ABB RobotStudio station: Train_assembly_setup_60.rsstn

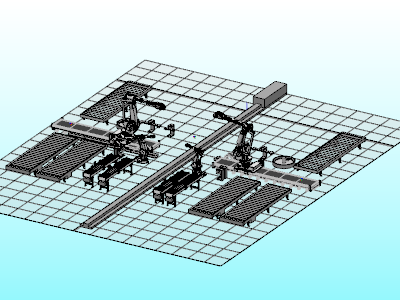
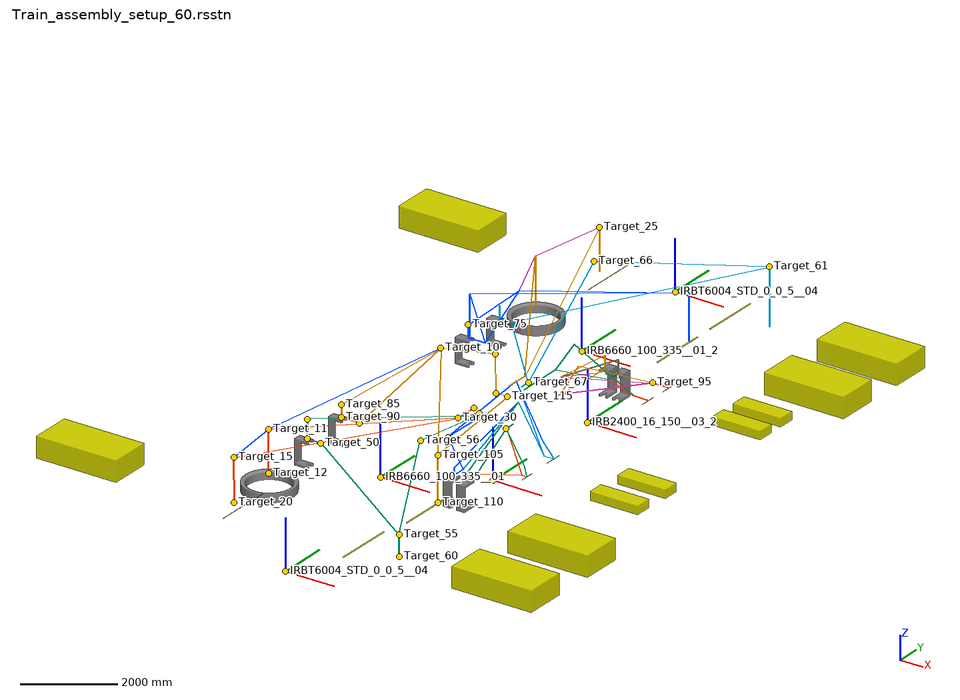
[picture v1: parts stored in the station drawn from their meshes, with robot base, taught points and paths (robot models come from the ABB library and are not in the file)]
Station Train_assembly_setup_60 (saved by RobotStudio 24.3.10958.1)
Controller Controller19, task T_ROB2: task frame (RAPID world) sits at (6880.03, 7396.16, 384.5) mm, rotated rx 0 ry 0 rz -90 deg in the station
Controller Controller19, task T_ROB1: task frame (RAPID world) sits at (6880.03, 7396.16, 384.5) mm, rotated rx 0 ry 0 rz -90 deg in the station
Controller Controller18, task T_ROB2: task frame (RAPID world) sits at (6882.77, -6739.06, 384.5) mm, rotated rx 0 ry 0 rz 90 deg in the station
Controller Controller18, task T_ROB1: task frame (RAPID world) sits at (6882.77, -6739.06, 384.5) mm, rotated rx 0 ry 0 rz 90 deg in the station
Controller Controller18
  mechanical unit ROB_1: IRB6660_100_335__01, 6 joints, base frame (0, 0, 0) mm
  mechanical unit TRACK_1: IRBT6004_STD_0_0_5__04, 1 joints, base frame (0, 0, 0) mm
  mechanical unit ROB_2: IRB2400_16_150__03, 6 joints, base frame (5338.88, -1522.95, -384.5) mm, rotated rx 0 ry 0 rz 0.09 deg
Controller Controller19
  mechanical unit ROB_1: IRB6660_100_335__01_2, 6 joints, base frame (0, 0, 0) mm
  mechanical unit TRACK_1: IRBT6004_STD_0_0_5__04_2, 1 joints, base frame (0, 0, 0) mm
  mechanical unit ROB_2: IRB2400_16_150__03_2, 6 joints, base frame (5457.45, 1561.32, -384.5) mm, rotated rx 0 ry 0 rz -0.15 deg
Layout (positions relative to the parent item):
  - train_body [part] at (-4902.1, 350, 1462.39) mm, rotated rx 90 ry 0 rz 90 deg, size 1000 x 1362.5 x 2750 mm
  - IRB6660_100_335__01 [mechanism, from %ABB.RobotStudio.Models.IRB6660%\IRB6660_100_335_G_01.rslib] at (6882.77, -3243.33, 384.5) mm, rotated rx 0 ry 0 rz 90 deg; joint values [0.0868, -0.0685, 0.1058, 0, 0.4178, 1.215] (rad or m)
  - IRBT6004_STD_0_0_5__04 [mechanism] at (7357.77, -7329.56, 0) mm, rotated rx 0 ry 0 rz 90 deg; joint values [3.4957] (rad or m)
      links: Base, Link1
  - IRB2400_16_150__03 [mechanism, from %ABB.RobotStudio.Models.IRB2400%\IRB2400_16_150_G_03.rslib] at (8405.72, -1400.18, 0) mm, rotated rx 0 ry 0 rz 90.09 deg; joint values [0, -0.2615, -0.2111, 0, 0.7347, 0] (rad or m)
  - toolHolder_2 [part] at (8688, -2615.24, 0) mm, rotated rx 0 ry 0 rz 180 deg, size 200 x 350 x 600 mm
  - toolHolder_3 [part] at (8343.34, -2615.24, 0) mm, rotated rx 0 ry 0 rz 180 deg, size 200 x 350 x 600 mm
  - toolHolder_5 [part] at (4986.26, -1820.5, 17.28) mm, rotated rx 0 ry 0 rz 90 deg, size 200 x 350 x 600 mm
  - toolHolder_6 [part] at (4986.26, -3034.43, 0) mm, rotated rx 0 ry 0 rz 90 deg, size 200 x 350 x 600 mm
  - Axel_pin [part] at (11460.69, -1282, 854.82) mm, size 562.7 x 211 x 211 mm
  - ToolHolder(wheel) [part] at (4900.07, -4399.05, 0) mm, size 1200 x 1193.4 x 200 mm
  - 1320_4800_h2 [part, from %ABB.RobotStudio.Models.Conveyors%\Conveyor 1320 4800 h2.rslib] at (701.25, 6246.74, 0) mm
  - 1320_4800_2 [part, from %ABB.RobotStudio.Models.Conveyors%\Conveyor 1320 4800 h2.rslib] at (13264.62, -5495.83, 0) mm, rotated rx 0 ry 0 rz 180 deg
  - 1320_4800_3 [part, from %ABB.RobotStudio.Models.Conveyors%\Conveyor 1320 4800 h2.rslib] at (13264.62, -3687.06, 0) mm, rotated rx 0 ry 0 rz 180 deg
  - Stack_tutorial_2 [part] at (8828.86, 5027.59, 1315.99) mm, rotated rx -90 ry 0 rz 0 deg, size 625 x 875 x 623.8 mm
  - Cow_Catcher [part] at (13797.89, -3839.41, 450.44) mm, rotated rx 0 ry 0 rz -90 deg, size 900 x 562.5 x 375 mm
  - Link [part] at (13394.81, -6331.06, 437.55) mm, rotated rx 90 ry 0 rz -90 deg, size 186.8 x 62.5 x 1937.5 mm
  - Arm_pin [part] at (10630.82, -2218.47, 824.2) mm, rotated rx 0 ry 0 rz 90 deg, size 126 x 162.5 x 125.8 mm
  - 400_guide [part, from %ABB.RobotStudio.Models.Conveyors%\Conveyor Guide 400.rslib] at (12859.46, 2271.9, 0) mm, rotated rx 0 ry 0 rz 180 deg
  - 400 [part, from %ABB.RobotStudio.Models.Conveyors%\Conveyor Guide 400.rslib] at (12859.46, -2034.23, 0) mm, rotated rx 0 ry 0 rz 180 deg
  - ZugSchlitten [mechanism] at (-2951.59, 0, 0) mm; joint values [0] (rad or m)
      links: L1, L2
  - MoveTrain_Wheel1 [smart component]
      signals: DI GetToWheel1
      connections:
        MoveTrain_Wheel1.GetToWheel1 -> PoseMover.Execute
    - PoseMover [smart component, from Components\PoseMover.rslib]
        properties: Mechanism=ZugSchlitten; Pose=2; Duration=2
  - Wheel_tool_smart [smart component] at (4882.6, -4404, 384.25) mm, rotated rx 180 ry 0 rz -0.66 deg
      signals: DI Wheel_Attach, DO Wheel_is_attached, DI findLocomotive
      connections:
        Attacher.Executed -> Wheel_tool_smart.Wheel_is_attached
        Wheel_tool_smart.Wheel_Attach -> LogicGate.InputA
        LogicGate.Output -> Detacher.Execute
        Attacher.Executed -> SetParent_2.Execute
        Detacher.Executed -> SetParent_3.Execute
        Detacher.Executed -> Attacher_2.Execute
        Wheel_tool_smart.Wheel_Attach -> ClosestObject.Execute
        ClosestObject.Executed -> Attacher.Execute
        Wheel_tool_smart.Wheel_Attach -> ClosestObject_2.Execute
        Attacher.Child => Detacher.Child
        Attacher.Child => SetParent_2.Child
        Attacher.Child => SetParent_3.Child
        Detacher.Child => Attacher_2.Child
        ClosestObject.ClosestObject => Attacher.Child
        ClosestObject.ReferenceObject => Attacher.Parent
        ClosestObject_2.ClosestObject => Attacher_2.Parent
    - WheelTool [mechanism] at (0, 0, 0) mm
        TCP WheelTool at (0, 0, 380) mm
        links: Tool_Wheel
    - Attacher [smart component, from Components\Attacher.rslib]
        properties: Parent=WheelTool; Flange=0; Child=Link_Tool_smart; Mount=false; Offset=[0 0 0]; Orientation=[0 0 0]
    - LogicGate [smart component, from Components\LogicGate.rslib]
        properties: Operator=NOT; Delay=0
    - Detacher [smart component, from Components\Detacher.rslib]
        properties: Child=Link_Tool_smart; KeepPosition=true
    - Attacher_2 [smart component, from Components\Attacher.rslib]
        properties: Parent=train_body; Flange=0; Child=Link_Tool_smart; Mount=false; Offset=[0 0 0]; Orientation=[0 0 0]
    - ClosestObject [smart component, from Components\ClosestObject.rslib]
        properties: ReferenceObject=Wheel_tool_smart; ReferencePoint=[0 0 0]; RootObject=(none); ClosestObject=Link_Tool_smart; ClosestPart=Tool_Link; Distance=0.444833038330078
    - ClosestObject_2 [smart component, from Components\ClosestObject.rslib]
        properties: ReferenceObject=L2; ReferencePoint=[0 0 0]; RootObject=(none); ClosestObject=train_body; ClosestPart=train_body; Distance=0
  - Wheel [part] at (3497.77, -6177.47, 411.44) mm, size 1122.9 x 1119.7 x 250 mm
  - Axel_Tool_smart [smart component] at (8343.34, -2684.49, 620.79) mm, rotated rx 180 ry 0 rz 0 deg
      signals: DI Grab_with_tool, DO partAttached
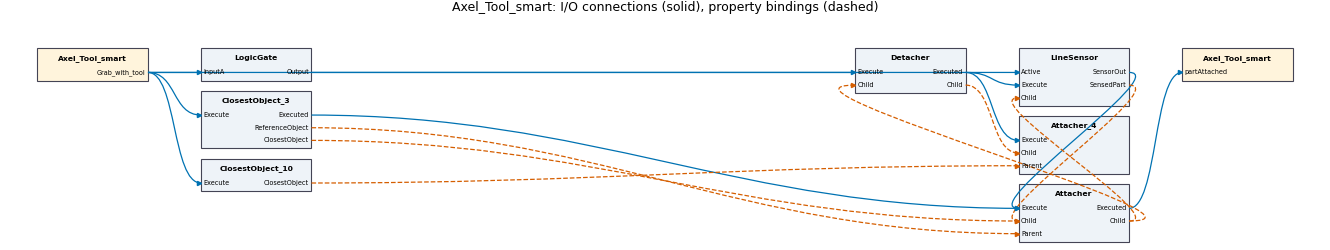
      connections:
        Axel_Tool_smart.Grab_with_tool -> LineSensor.Active
        LineSensor.SensorOut -> Attacher.Execute
        Axel_Tool_smart.Grab_with_tool -> LogicGate.InputA
        LogicGate.Output -> Detacher.Execute
        Detacher.Executed -> SetParent_4.Execute
        Attacher.Executed -> Axel_Tool_smart.partAttached
        Axel_Tool_smart.Grab_with_tool -> ClosestObject_3.Execute
        ClosestObject_3.Executed -> Attacher.Execute
        Detacher.Executed -> Attacher_4.Execute
        Axel_Tool_smart.Grab_with_tool -> ClosestObject_10.Execute
        LineSensor.SensedPart => Attacher.Child
        Attacher.Child => Detacher.Child
        Attacher.Child => SetParent_4.Child
        ClosestObject_3.ReferenceObject => Attacher.Parent
        ClosestObject_3.ClosestObject => Attacher.Child
        Detacher.Child => Attacher_4.Child
        ClosestObject_10.ClosestObject => Attacher_4.Parent
    - AxelTool [mechanism] at (0, 9.42, 0) mm
        TCP AxelTool at (0, 0, 262.49) mm
        links: Tool_Axel_pin
    - Detacher [smart component, from Components\Detacher.rslib]
        properties: Child=Pin_Tool_smart; KeepPosition=true
    - LogicGate [smart component, from Components\LogicGate.rslib]
        properties: Operator=NOT; Delay=0
    - Attacher [smart component, from Components\Attacher.rslib]
        properties: Parent=Axel_Tool_smart; Flange=0; Child=Pin_Tool_smart; Mount=false; Offset=[0 0 0]; Orientation=[0 0 0]
    - ClosestObject_3 [smart component, from Components\ClosestObject.rslib]
        properties: ReferenceObject=Axel_Tool_smart; ReferencePoint=[0 0 0]; RootObject=(none); ClosestObject=Pin_Tool_smart; ClosestPart=Tool_Arm_pin; Distance=0.139682907104492
    - Attacher_4 [smart component, from Components\Attacher.rslib]
        properties: Parent=(none); Flange=0; Child=Pin_Tool_smart; Mount=false; Offset=[0 0 0]; Orientation=[0 0 0]
    - ClosestObject_10 [smart component, from Components\ClosestObject.rslib]
        properties: ReferenceObject=L2; ReferencePoint=[0 0 0]; RootObject=(none); ClosestObject=(none); ClosestPart=(none); Distance=0
  - AttachTool_Rob1 [smart component] at (6695.48, -1090.62, 2469) mm, rotated rx 121.63 ry 17.56 rz -164.5 deg
      signals: DI AttachTool, DO ToolAttached
      connections:
        AttachTool_Rob1.AttachTool -> ClosestObject.Execute
        ClosestObject.Executed -> Attacher.Execute
        AttachTool_Rob1.AttachTool -> LogicGate.InputA
        LogicGate.Output -> Detacher.Execute
        Attacher.Executed -> AttachTool_Rob1.ToolAttached
        ClosestObject.ClosestObject => Attacher.Child
        Attacher.Child => Detacher.Child
    - ClosestObject [smart component, from Components\ClosestObject.rslib]
        properties: ReferenceObject=IRB6660_100_335__01; ReferencePoint=[7.13389 -0.654994 0.85]; RootObject=(none); ClosestObject=Axel_Tool_smart; ClosestPart=Tool_Axel_pin; Distance=0.924461853027344
    - Attacher [smart component, from Components\Attacher.rslib]
        properties: Parent=IRB6660_100_335__01; Flange=0; Child=Axel_Tool_smart; Mount=false; Offset=[0 0 0]; Orientation=[0 0 0]
    - LogicGate [smart component, from Components\LogicGate.rslib]
        properties: Operator=NOT; Delay=0
    - Detacher [smart component, from Components\Detacher.rslib]
        properties: Child=Axel_Tool_smart; KeepPosition=true
  - AttachTool_Rob2 [smart component] at (8404.6, -698.88, 1543.74) mm, rotated rx 180 ry 60 rz -89.91 deg
      signals: DI AttachTool, DO ToolAttached
      connections:
        AttachTool_Rob2.AttachTool -> ClosestObject.Execute
        ClosestObject.Executed -> Attacher.Execute
        AttachTool_Rob2.AttachTool -> LogicGate.InputA
        LogicGate.Output -> Detacher.Execute
        Attacher.Executed -> AttachTool_Rob2.ToolAttached
        ClosestObject.ClosestObject => Attacher.Child
        Attacher.Child => Detacher.Child
    - ClosestObject [smart component, from Components\ClosestObject.rslib]
        properties: ReferenceObject=IRB2400_16_150__03; ReferencePoint=[7.483895 -1.376883 0.85]; RootObject=(none); ClosestObject=Axel_Tool_smart; ClosestPart=Tool_Axel_pin; Distance=0.745236877441406
    - Attacher [smart component, from Components\Attacher.rslib]
        properties: Parent=IRB2400_16_150__03; Flange=0; Child=Axel_Tool_smart; Mount=false; Offset=[0 0 0]; Orientation=[0 0 0]
    - LogicGate [smart component, from Components\LogicGate.rslib]
        properties: Operator=NOT; Delay=0
    - Detacher [smart component, from Components\Detacher.rslib]
        properties: Child=Axel_Tool_smart; KeepPosition=true
  - MoveTrain_Wheel2 [smart component]
      signals: DI GetToWheel2
      connections:
        MoveTrain_Wheel2.GetToWheel2 -> PoseMover.Execute
    - PoseMover [smart component, from Components\PoseMover.rslib]
        properties: Mechanism=ZugSchlitten; Pose=3; Duration=1
  - Locomotive [smart component] at (-3926.39, 500, 862.39) mm
  - SpawnWheel [smart component]
      signals: DO volumeerkannt, DI spanw, DI diDeque
      connections:
        VolumeSensor.SensorOut -> LogicGate.InputA
        LineSensor_2.SensorOut -> LogicGate_2.InputA
        LogicGate_2.Output -> LinearMover.Execute
        Source.Executed -> Queue_2.Enqueue
        LogicGate.Output -> Source.Execute
        SpawnWheel.diDeque -> Queue_2.Dequeue
        SpawnWheel.spanw -> Source.Execute
        Source.Copy => Queue_2.Back
    - Source [smart component, from Components\Source.rslib]
        properties: Source=Wheel; Copy=(none); Parent=(none); Position=[1.2 -6.177465 0.41144]; Orientation=[0 0 0]; Transient=false; PhysicsBehavior=-1
    - Queue_2 [smart component, from Components\Queue.rslib]
        properties: Back=(none); Front=(none); Queue={1d260e56-3a9b-4089-bc8a-9b7fc13f89e8};{5a10ac6e-8e6d-4320-b1fc-87ca64eb2ab9}; NumberOfObjects=2
    - LinearMover [smart component, from Components\LinearMover.rslib]
        properties: Object=Queue_2; Direction=[1 0 0]; Speed=0.8; Reference=Global; ReferenceObject=(none)
    - LineSensor_2 [smart component, from Components\LineSensor.rslib]
        properties: Start=[5.47 -6.89178 0.5]; End=[5.47 -5.45178 0.5]; Length=1.44; Radius=0.00524017467248908; Tag=(none); SensedPart=(none); SensedPoint=[0 0 0]
      - _sensorPart_ [part], size 10.5 x 1440 x 10.5 mm
    - VolumeSensor [smart component, from Components\VolumeSensor.rslib]
        properties: CornerPoint=[0.761246 -6.83178 0.55]; Orientation=[0 0 0]; Length=2; Width=1; Height=0.5; Tag=(none); PartialHit=true; SensedPart=(none)
      - _sensorPart_ [part], size 2000 x 1000 x 500 mm
    - LogicGate [smart component, from Components\LogicGate.rslib]
        properties: Operator=NOT; Delay=0
    - LogicGate_2 [smart component, from Components\LogicGate.rslib]
        properties: Operator=NOT; Delay=0
  - SpawnAxel [smart component]
      signals: DO volumeerkannt, DI spanw, DI diDeque
      connections:
        VolumeSensor.SensorOut -> LogicGate.InputA
        LineSensor_2.SensorOut -> LogicGate_2.InputA
        LogicGate_2.Output -> LinearMover.Execute
        Source.Executed -> Queue_2.Enqueue
        LogicGate.Output -> Source.Execute
        SpawnAxel.diDeque -> Queue_2.Dequeue
        Source.Copy => Queue_2.Back
    - Source [smart component, from Components\Source.rslib]
        properties: Source=Axel_pin; Copy=(none); Parent=(none); Position=[12.5 -1.280871 0.854819]; Orientation=[0 0 0]; Transient=false; PhysicsBehavior=-1
    - Queue_2 [smart component, from Components\Queue.rslib]
        properties: Back=(none); Front=(none); Queue={1d260e56-3a9b-4089-bc8a-9b7fc13f89e8}; NumberOfObjects=1
    - LinearMover [smart component, from Components\LinearMover.rslib]
        properties: Object=Queue_2; Direction=[-1 0 0]; Speed=0.5; Reference=Global; ReferenceObject=(none)
    - LineSensor_2 [smart component, from Components\LineSensor.rslib]
        properties: Start=[9.859459 -1.543182 0.86]; End=[9.859459 -1.100182 0.86]; Length=0.443; Radius=0.00524017467248908; Tag=(none); SensedPart=(none); SensedPoint=[0 0 0]
      - _sensorPart_ [part], size 10.5 x 443 x 10.5 mm
    - VolumeSensor [smart component, from Components\VolumeSensor.rslib]
        properties: CornerPoint=[11.6 -1.5 0.86]; Orientation=[0 0 0]; Length=1.2; Width=0.4; Height=0.2; Tag=(none); PartialHit=true; SensedPart=(none)
      - _sensorPart_ [part], size 1200 x 400 x 200 mm
    - LogicGate [smart component, from Components\LogicGate.rslib]
        properties: Operator=NOT; Delay=0
    - LogicGate_2 [smart component, from Components\LogicGate.rslib]
        properties: Operator=NOT; Delay=0
  - IRB2400_16_150__03_2 [mechanism, from %ABB.RobotStudio.Models.IRB2400%\IRB2400_16_150_G_03.rslib] at (8441.35, 1938.71, 0) mm, rotated rx 0 ry 0 rz -90.15 deg; joint values [0, -0.2615, -0.2111, 0, 0.7347, 0] (rad or m)
  - IRBT6004_STD_0_0_5__04_2 [mechanism] at (6405.03, 7986.66, 0) mm, rotated rx 0 ry 0 rz -90 deg; joint values [3.4275] (rad or m)
      links: Base, Link1
  - IRB6660_100_335__01_2 [mechanism, from %ABB.RobotStudio.Models.IRB6660%\IRB6660_100_335_G_01.rslib] at (6880.03, 3968.65, 384.5) mm, rotated rx 0 ry 0 rz -90 deg; joint values [0, -0.2199, -0.1274, 0, 0.651, 0] (rad or m)
  - 1320_4800_4 [part, from %ABB.RobotStudio.Models.Conveyors%\Conveyor 1320 4800 h2.rslib] at (701.25, -6831.78, 0) mm
  - ToolHolder(wheel)_2 [part] at (4900.07, 5155.46, 0) mm, size 1200 x 1193.4 x 200 mm
  - toolHolder_7 [part] at (4986.26, 3849.13, 0) mm, rotated rx 0 ry 0 rz 90 deg, size 200 x 350 x 600 mm
  - toolHolder_8 [part] at (4986.26, 2721.93, 17.28) mm, rotated rx 0 ry 0 rz 90 deg, size 200 x 350 x 600 mm
  - Wheel_tool_smart_2 [smart component] at (4882.6, 5151.99, 384.25) mm, rotated rx -180 ry 0 rz -0.66 deg
      signals: DI Wheel_Attach, DO Wheel_is_attached
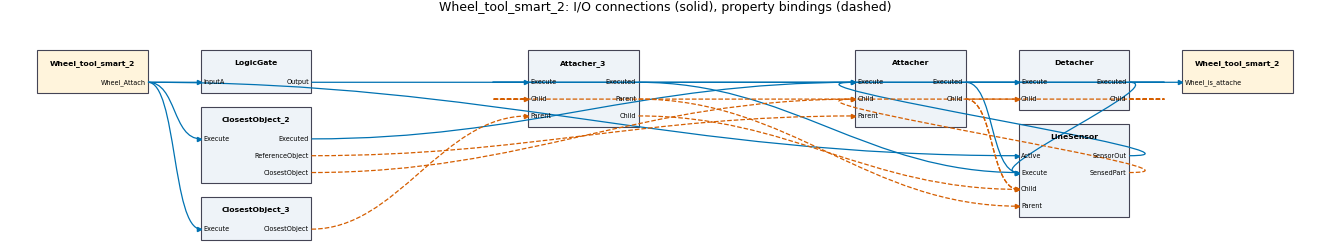
      connections:
        Wheel_tool_smart_2.Wheel_Attach -> LineSensor.Active
        LineSensor.SensorOut -> Attacher.Execute
        Attacher.Executed -> Wheel_tool_smart_2.Wheel_is_attached
        Wheel_tool_smart_2.Wheel_Attach -> LogicGate.InputA
        LogicGate.Output -> Detacher.Execute
        Attacher.Executed -> ?.Execute
        Detacher.Executed -> SetParent_3.Execute
        Wheel_tool_smart_2.Wheel_Attach -> ClosestObject_2.Execute
        ClosestObject_2.Executed -> Attacher.Execute
        Detacher.Executed -> Attacher_3.Execute
        Wheel_tool_smart_2.Wheel_Attach -> ClosestObject_3.Execute
        Attacher_3.Executed -> SetParent.Execute
        LineSensor.SensedPart => Attacher.Child
        Attacher.Child => Detacher.Child
        Attacher.Child => ?.Child
        Attacher.Child => SetParent_3.Child
        ClosestObject_2.ReferenceObject => Attacher.Parent
        ClosestObject_2.ClosestObject => Attacher.Child
        Detacher.Child => Attacher_3.Child
        ClosestObject_3.ClosestObject => Attacher_3.Parent
        Attacher_3.Parent => SetParent.Parent
        Attacher_3.Child => SetParent.Child
    - WheelTool [mechanism] at (11.79, -0.14, 0) mm
        TCP WheelTool at (0, 0, 380) mm
        links: Tool_Wheel
    - Attacher [smart component, from Components\Attacher.rslib]
        properties: Parent=WheelTool; Flange=0; Child=Link_Tool_smart_2; Mount=false; Offset=[0 0 0]; Orientation=[0 0 0]
    - LogicGate [smart component, from Components\LogicGate.rslib]
        properties: Operator=NOT; Delay=0
    - Detacher [smart component, from Components\Detacher.rslib]
        properties: Child=Link_Tool_smart_2; KeepPosition=true
    - ClosestObject_2 [smart component, from Components\ClosestObject.rslib]
        properties: ReferenceObject=Wheel_tool_smart_2; ReferencePoint=[0 0 0]; RootObject=(none); ClosestObject=Link_Tool_smart_2; ClosestPart=Tool_Link; Distance=0.391564422607422
    - Attacher_3 [smart component, from Components\Attacher.rslib]
        properties: Parent=train_body; Flange=0; Child=Link_Tool_smart_2; Mount=false; Offset=[0 0 0]; Orientation=[0 0 0]
    - ClosestObject_3 [smart component, from Components\ClosestObject.rslib]
        properties: ReferenceObject=L2; ReferencePoint=[0 0 0]; RootObject=(none); ClosestObject=train_body; ClosestPart=train_body; Distance=1.51384008789063
  - toolHolder_10 [part] at (8343.34, 3102.04, 0) mm, size 200 x 350 x 600 mm
  - 400_2 [part, from %ABB.RobotStudio.Models.Conveyors%\Conveyor Guide 400.rslib] at (12859.46, -1103.18, 0) mm, rotated rx 0 ry 0 rz 180 deg
  - SpawnAxel_2 [smart component]
      signals: DO volumeerkannt, DI spanw, DI diDeque
      connections:
        VolumeSensor.SensorOut -> LogicGate.InputA
        LineSensor_2.SensorOut -> LogicGate_2.InputA
        LogicGate_2.Output -> LinearMover.Execute
        Source.Executed -> Queue_2.Enqueue
        LogicGate.Output -> Source.Execute
        SpawnAxel_2.diDeque -> Queue_2.Dequeue
        SpawnAxel_2.spanw -> Source.Execute
        VolumeSensor.SensorOut -> SpawnAxel_2.volumeerkannt
        Source.Copy => Queue_2.Back
    - Source [smart component, from Components\Source.rslib]
        properties: Source=Axel_pin_2; Copy=(none); Parent=(none); Position=[12.5 2.071151 0.854819]; Orientation=[0 0 0]; Transient=false; PhysicsBehavior=-1
    - Queue_2 [smart component, from Components\Queue.rslib]
        properties: Back=(none); Front=(none); Queue={1d260e56-3a9b-4089-bc8a-9b7fc13f89e8};{68ae6273-f876-46ed-a841-c22bc3c7f170}; NumberOfObjects=1
    - LinearMover [smart component, from Components\LinearMover.rslib]
        properties: Object=Queue_2; Direction=[-1 0 0]; Speed=0.5; Reference=Global; ReferenceObject=(none)
    - LineSensor_2 [smart component, from Components\LineSensor.rslib]
        properties: Start=[9.859459 1.8769 0.84]; End=[9.859459 2.2749 0.84]; Length=0.398; Radius=0.00524017467248908; Tag=(none); SensedPart=(none); SensedPoint=[0 0 0]
      - _sensorPart_ [part], size 10.5 x 398 x 10.5 mm
    - VolumeSensor [smart component, from Components\VolumeSensor.rslib]
        properties: CornerPoint=[11.617459 1.8719 0.86]; Orientation=[0 0 0]; Length=1.2; Width=0.4; Height=0.2; Tag=(none); PartialHit=true; SensedPart=(none)
      - _sensorPart_ [part], size 1200 x 400 x 200 mm
    - LogicGate [smart component, from Components\LogicGate.rslib]
        properties: Operator=NOT; Delay=0
    - LogicGate_2 [smart component, from Components\LogicGate.rslib]
        properties: Operator=NOT; Delay=0
  - Axel_pin_2 [part] at (11364, 2071.15, 854.82) mm, size 562.7 x 211 x 211 mm
  - Axel_Tool_smart_2 [smart component] at (8343.34, 3189.01, 620.79) mm, rotated rx 180 ry 0 rz 0 deg
      signals: DI Grab_with_tool, DO partAttached
      connections:
        Axel_Tool_smart_2.Grab_with_tool -> LineSensor.Active
        LineSensor.SensorOut -> Attacher.Execute
        Axel_Tool_smart_2.Grab_with_tool -> LogicGate.InputA
        LogicGate.Output -> Detacher.Execute
        Detacher.Executed -> SetParent_4.Execute
        Attacher.Executed -> Axel_Tool_smart_2.partAttached
        Axel_Tool_smart_2.Grab_with_tool -> ClosestObject_4.Execute
        ClosestObject_4.Executed -> Attacher.Execute
        Detacher.Executed -> Attacher_5.Execute
        Axel_Tool_smart_2.Grab_with_tool -> ClosestObject_11.Execute
        LineSensor.SensedPart => Attacher.Child
        Attacher.Child => Detacher.Child
        Attacher.Child => SetParent_4.Child
        ClosestObject_4.ReferenceObject => Attacher.Parent
        ClosestObject_4.ClosestObject => Attacher.Child
        Detacher.Child => Attacher_5.Child
        ClosestObject_11.ClosestObject => Attacher_5.Parent
    - AxelTool [mechanism] at (0, 9.42, 0) mm
        TCP AxelTool at (0, 0, 262.49) mm
        links: Tool_Axel_pin
    - Detacher [smart component, from Components\Detacher.rslib]
        properties: Child=toolHolder_10; KeepPosition=true
    - LogicGate [smart component, from Components\LogicGate.rslib]
        properties: Operator=NOT; Delay=0
    - Attacher [smart component, from Components\Attacher.rslib]
        properties: Parent=Axel_Tool_smart_2; Flange=0; Child=toolHolder_10; Mount=false; Offset=[0 0 0]; Orientation=[0 0 0]
    - ClosestObject_4 [smart component, from Components\ClosestObject.rslib]
        properties: ReferenceObject=Axel_Tool_smart_2; ReferencePoint=[0 0 0]; RootObject=(none); ClosestObject=toolHolder_10; ClosestPart=toolHolder_10; Distance=0
    - Attacher_5 [smart component, from Components\Attacher.rslib]
        properties: Parent=train_body; Flange=0; Child=toolHolder_10; Mount=false; Offset=[0 0 0]; Orientation=[0 0 0]
    - ClosestObject_11 [smart component, from Components\ClosestObject.rslib]
        properties: ReferenceObject=L2; ReferencePoint=[0 0 0]; RootObject=(none); ClosestObject=train_body; ClosestPart=train_body; Distance=1.51384008789063
  - AttachTool_Rob4 [smart component] at (8508.36, -848.72, 1842.51) mm, rotated rx 14.33 ry -9.97 rz 155.57 deg
      signals: DI AttachTool, DO ToolAttached
      connections:
        AttachTool_Rob4.AttachTool -> ClosestObject.Execute
        ClosestObject.Executed -> Attacher.Execute
        AttachTool_Rob4.AttachTool -> LogicGate.InputA
        LogicGate.Output -> Detacher.Execute
        Attacher.Executed -> AttachTool_Rob4.ToolAttached
        ClosestObject.ClosestObject => Attacher.Child
        Attacher.Child => Detacher.Child
    - ClosestObject [smart component, from Components\ClosestObject.rslib]
        properties: ReferenceObject=IRB2400_16_150__03_2; ReferencePoint=[7.483895 1.442587 0.85]; RootObject=(none); ClosestObject=toolHolder_10; ClosestPart=toolHolder_10; Distance=0.689487548828125
    - Attacher [smart component, from Components\Attacher.rslib]
        properties: Parent=IRB2400_16_150__03_2; Flange=0; Child=toolHolder_10; Mount=false; Offset=[0 0 0]; Orientation=[0 0 0]
    - LogicGate [smart component, from Components\LogicGate.rslib]
        properties: Operator=NOT; Delay=0
    - Detacher [smart component, from Components\Detacher.rslib]
        properties: Child=toolHolder_10; KeepPosition=true
  - AttachTool_Rob3 [smart component] at (8508.36, -848.72, 1842.51) mm, rotated rx 14.33 ry -9.97 rz 155.57 deg
      signals: DI AttachTool, DO ToolAttached
      connections:
        AttachTool_Rob3.AttachTool -> ClosestObject.Execute
        ClosestObject.Executed -> Attacher.Execute
        AttachTool_Rob3.AttachTool -> LogicGate.InputA
        LogicGate.Output -> Detacher.Execute
        Attacher.Executed -> AttachTool_Rob3.ToolAttached
        ClosestObject.ClosestObject => Attacher.Child
        Attacher.Child => Detacher.Child
    - ClosestObject [smart component, from Components\ClosestObject.rslib]
        properties: ReferenceObject=IRB6660_100_335__01_2; ReferencePoint=[4.894392 5.151995 0.65291]; RootObject=(none); ClosestObject=Pin_Tool_smart2; ClosestPart=Tool_Arm_pin; Distance=0.77755078125
    - Attacher [smart component, from Components\Attacher.rslib]
        properties: Parent=IRB6660_100_335__01_2; Flange=0; Child=Pin_Tool_smart2; Mount=false; Offset=[0 0 0]; Orientation=[0 0 0]
    - LogicGate [smart component, from Components\LogicGate.rslib]
        properties: Operator=NOT; Delay=0
    - Detacher [smart component, from Components\Detacher.rslib]
        properties: Child=Pin_Tool_smart2; KeepPosition=true
  - Wheel_2 [part] at (3426.57, 6899.85, 411.8) mm, size 1122.9 x 1119.7 x 250 mm
  - SpawnWheel_2 [smart component]
      signals: DO volumeerkannt, DI spanw, DI diDeque
      connections:
        VolumeSensor.SensorOut -> LogicGate.InputA
        LineSensor_2.SensorOut -> LogicGate_2.InputA
        LogicGate_2.Output -> LinearMover.Execute
        Source.Executed -> Queue_2.Enqueue
        LogicGate.Output -> Source.Execute
        SpawnWheel_2.diDeque -> Queue_2.Dequeue
        SpawnWheel_2.spanw -> Source.Execute
        Source.Copy => Queue_2.Back
    - Source [smart component, from Components\Source.rslib]
        properties: Source=Wheel_2; Copy=(none); Parent=(none); Position=[1.8 6.899851 0.411803]; Orientation=[0 0 0]; Transient=false; PhysicsBehavior=-1
    - Queue_2 [smart component, from Components\Queue.rslib]
        properties: Back=(none); Front=(none); Queue={1d260e56-3a9b-4089-bc8a-9b7fc13f89e8}; NumberOfObjects=1
    - LinearMover [smart component, from Components\LinearMover.rslib]
        properties: Object=Queue_2; Direction=[1 0 0]; Speed=0.8; Reference=Global; ReferenceObject=(none)
    - LineSensor_2 [smart component, from Components\LineSensor.rslib]
        properties: Start=[5.47 6.186738 0.5]; End=[5.47 7.626738 0.5]; Length=1.44; Radius=0.00524017467248908; Tag=(none); SensedPart=(none); SensedPoint=[0 0 0]
      - _sensorPart_ [part], size 10.5 x 1440 x 10.5 mm
    - VolumeSensor [smart component, from Components\VolumeSensor.rslib]
        properties: CornerPoint=[0.577246 6.4 0.471]; Orientation=[0 0 0]; Length=2; Width=1; Height=0.5; Tag=(none); PartialHit=true; SensedPart=(none)
      - _sensorPart_ [part], size 2000 x 1000 x 500 mm
    - LogicGate [smart component, from Components\LogicGate.rslib]
        properties: Operator=NOT; Delay=0
    - LogicGate_2 [smart component, from Components\LogicGate.rslib]
        properties: Operator=NOT; Delay=0
  - 1320_4800_5 [part, from %ABB.RobotStudio.Models.Conveyors%\Conveyor 1320 4800 h2.rslib] at (13264.62, 7587.02, 0) mm, rotated rx 0 ry 0 rz 180 deg
  - Link_Tool_smart [smart component]
      signals: DI Link_Attach, DO Link_is_attached
      connections:
        Link_Tool_smart.Link_Attach -> ClosestObject.Execute
        ClosestObject.Executed -> Attacher.Execute
        Link_Tool_smart.Link_Attach -> LogicGate.InputA
        LogicGate.Output -> Detacher.Execute
        Detacher.Executed -> Attacher_2.Execute
        Attacher.Executed -> Link_Tool_smart.Link_is_attached
        Link_Tool_smart.Link_Attach -> ClosestObject_4.Execute
        ClosestObject.ReferenceObject => Attacher.Parent
        ClosestObject.ClosestObject => Attacher.Child
        Attacher.Child => Detacher.Child
        Detacher.Child => Attacher_2.Child
        ClosestObject_4.ClosestObject => Attacher_2.Parent
    - LinkTool [mechanism] at (4906.26, -3034.43, 624.04) mm, rotated rx 180 ry 0 rz 0 deg
        TCP LinkTool at (0, 0, 170) mm
        links: Tool_Link
    - ClosestObject [smart component, from Components\ClosestObject.rslib]
        properties: ReferenceObject=Link_Tool_smart; ReferencePoint=[0 0 0]; RootObject=(none); ClosestObject=Wheel_tool_smart; ClosestPart=Tool_Wheel; Distance=0.444832855224609
    - Attacher [smart component, from Components\Attacher.rslib]
        properties: Parent=Link_Tool_smart; Flange=0; Child=Wheel_tool_smart; Mount=false; Offset=[0 0 0]; Orientation=[0 0 0]
    - LogicGate [smart component, from Components\LogicGate.rslib]
        properties: Operator=NOT; Delay=0
    - Detacher [smart component, from Components\Detacher.rslib]
        properties: Child=Wheel_tool_smart; KeepPosition=true
    - Attacher_2 [smart component, from Components\Attacher.rslib]
        properties: Parent=(none); Flange=0; Child=Wheel_tool_smart; Mount=false; Offset=[0 0 0]; Orientation=[0 0 0]
    - ClosestObject_4 [smart component, from Components\ClosestObject.rslib]
        properties: ReferenceObject=L2; ReferencePoint=[0 0 0]; RootObject=(none); ClosestObject=(none); ClosestPart=(none); Distance=0
  - Pin_Tool_smart [smart component]
      signals: DI AttachPin, DO Pin_Attached
      connections:
        Pin_Tool_smart.AttachPin -> ClosestObject.Execute
        ClosestObject.Executed -> Attacher.Execute
        Pin_Tool_smart.AttachPin -> LogicGate.InputA
        LogicGate.Output -> Detacher.Execute
        Detacher.Executed -> Attacher_2.Execute
        Attacher.Executed -> Pin_Tool_smart.Pin_Attached
        Pin_Tool_smart.AttachPin -> ClosestObject_8.Execute
        ClosestObject.ReferenceObject => Attacher.Parent
        ClosestObject.ClosestObject => Attacher.Child
        Attacher.Child => Detacher.Child
        Detacher.Child => Attacher_2.Child
        ClosestObject_8.ClosestObject => Attacher_2.Parent
    - PinTool [mechanism] at (8688, -2695.24, 620.9) mm, rotated rx 180 ry 0 rz 0 deg
        TCP PinTool at (0, 0, 137.35) mm
        links: Tool_Arm_pin
    - ClosestObject [smart component, from Components\ClosestObject.rslib]
        properties: ReferenceObject=Pin_Tool_smart; ReferencePoint=[0 0 0]; RootObject=(none); ClosestObject=Axel_Tool_smart; ClosestPart=Tool_Axel_pin; Distance=0.139682907104492
    - Attacher [smart component, from Components\Attacher.rslib]
        properties: Parent=Pin_Tool_smart; Flange=0; Child=Axel_Tool_smart; Mount=false; Offset=[0 0 0]; Orientation=[0 0 0]
    - LogicGate [smart component, from Components\LogicGate.rslib]
        properties: Operator=NOT; Delay=0
    - Detacher [smart component, from Components\Detacher.rslib]
        properties: Child=Axel_Tool_smart; KeepPosition=true
    - Attacher_2 [smart component, from Components\Attacher.rslib]
        properties: Parent=(none); Flange=0; Child=Axel_Tool_smart; Mount=false; Offset=[0 0 0]; Orientation=[0 0 0]
    - ClosestObject_8 [smart component, from Components\ClosestObject.rslib]
        properties: ReferenceObject=L2; ReferencePoint=[0 0 0]; RootObject=(none); ClosestObject=(none); ClosestPart=(none); Distance=0
  - MoveTrain_Pin1 [smart component]
      signals: DI Move_to_pin1
      connections:
        MoveTrain_Pin1.Move_to_pin1 -> PoseMover.Execute
    - PoseMover [smart component, from Components\PoseMover.rslib]
        properties: Mechanism=ZugSchlitten; Pose=4; Duration=1
  - SpawnPin [smart component] at (0, -400, 0) mm
      signals: DO volumeerkannt, DI spanw, DI diDeque
      connections:
        VolumeSensor.SensorOut -> LogicGate.InputA
        LineSensor_2.SensorOut -> LogicGate_2.InputA
        LogicGate_2.Output -> LinearMover.Execute
        Source.Executed -> Queue_2.Enqueue
        LogicGate.Output -> Source.Execute
        SpawnPin.diDeque -> Queue_2.Dequeue
        Source.Copy => Queue_2.Back
    - Source [smart component, from Components\Source.rslib]
        properties: Source=Arm_pin; Copy=(none); Parent=(none); Position=[12.6 -2.218466 0.824201]; Orientation=[0 0 1.5707963267949]; Transient=false; PhysicsBehavior=-1
    - Queue_2 [smart component, from Components\Queue.rslib]
        properties: Back=(none); Front=(none); Queue={1d260e56-3a9b-4089-bc8a-9b7fc13f89e8}; NumberOfObjects=1
    - LinearMover [smart component, from Components\LinearMover.rslib]
        properties: Object=Queue_2; Direction=[-1 0 0]; Speed=0.5; Reference=Global; ReferenceObject=(none)
    - LineSensor_2 [smart component, from Components\LineSensor.rslib]
        properties: Start=[9.84 -1.633232 0.82]; End=[9.84 -2 0.82]; Length=0.366768; Radius=0.00524017467248908; Tag=(none); SensedPart=(none); SensedPoint=[0 0 0]
      - _sensorPart_ [part], size 10.5 x 366.8 x 10.5 mm
    - VolumeSensor [smart component, from Components\VolumeSensor.rslib]
        properties: CornerPoint=[11.56 -2.03 0.85]; Orientation=[0 0 0]; Length=1.2; Width=0.4; Height=0.2; Tag=(none); PartialHit=true; SensedPart=(none)
      - _sensorPart_ [part], size 1200 x 400 x 200 mm
    - LogicGate [smart component, from Components\LogicGate.rslib]
        properties: Operator=NOT; Delay=0
    - LogicGate_2 [smart component, from Components\LogicGate.rslib]
        properties: Operator=NOT; Delay=0
  - SpawnLink [smart component] at (10414.69, 0, 0) mm
      signals: DO volumeerkannt, DI spanw, DI diDeque
      connections:
        VolumeSensor.SensorOut -> LogicGate.InputA
        LineSensor_2.SensorOut -> LogicGate_2.InputA
        LogicGate_2.Output -> LinearMover.Execute
        Source.Executed -> Queue_2.Enqueue
        LogicGate.Output -> Source.Execute
        SpawnLink.diDeque -> Queue_2.Dequeue
        SpawnLink.spanw -> Source.Execute
        Source.Copy => Queue_2.Back
    - Source [smart component, from Components\Source.rslib]
        properties: Source=Link; Copy=(none); Parent=(none); Position=[11.5 -6.331 0.43755]; Orientation=[1.5707963267949 0 -1.5707963267949]; Transient=false; PhysicsBehavior=-1
    - Queue_2 [smart component, from Components\Queue.rslib]
        properties: Back=(none); Front=(none); Queue={1d260e56-3a9b-4089-bc8a-9b7fc13f89e8};{5a10ac6e-8e6d-4320-b1fc-87ca64eb2ab9};{339d23b8-4dd4-4c1e-9a58-b77691da5f86}; NumberOfObjects=1
    - LinearMover [smart component, from Components\LinearMover.rslib]
        properties: Object=Queue_2; Direction=[-1 0 0]; Speed=0.5; Reference=Global; ReferenceObject=(none)
    - LineSensor_2 [smart component, from Components\LineSensor.rslib] at (-7385.86, 0, -29.99) mm
        properties: Start=[5.47 -6.89178 0.5]; End=[5.47 -5.45178 0.5]; Length=1.44; Radius=0.0131004366812227; Tag=(none); SensedPart=(none); SensedPoint=[0 0 0]
      - _sensorPart_ [part], size 26.2 x 1440 x 26.2 mm
    - VolumeSensor [smart component, from Components\VolumeSensor.rslib]
        properties: CornerPoint=[0.761246486480401 -6.83178 0.49]; Orientation=[0 0 0]; Length=2; Width=1; Height=0.5; Tag=(none); PartialHit=true; SensedPart=(none)
      - _sensorPart_ [part], size 2000 x 1000 x 500 mm
    - LogicGate [smart component, from Components\LogicGate.rslib]
        properties: Operator=NOT; Delay=0
    - LogicGate_2 [smart component, from Components\LogicGate.rslib]
        properties: Operator=NOT; Delay=0
  - MoveTrain_Pin2 [smart component]
      signals: DI Get_to_Pin2
      connections:
        MoveTrain_Pin2.Get_to_Pin2 -> PoseMover.Execute
    - PoseMover [smart component, from Components\PoseMover.rslib]
        properties: Mechanism=ZugSchlitten; Pose=5; Duration=1
  - Link_Tool_smart_2 [smart component] at (4906.26, 3849.13, 626.19) mm
      signals: DI Link_Attach, DO Link_is_attached
      connections:
        Link_Tool_smart_2.Link_Attach -> ClosestObject.Execute
        ClosestObject.Executed -> Attacher.Execute
        Link_Tool_smart_2.Link_Attach -> LogicGate.InputA
        LogicGate.Output -> Detacher.Execute
        Detacher.Executed -> Attacher_2.Execute
        Attacher.Executed -> Link_Tool_smart_2.Link_is_attached
        Link_Tool_smart_2.Link_Attach -> ClosestObject_5.Execute
        ClosestObject.ReferenceObject => Attacher.Parent
        ClosestObject.ClosestObject => Attacher.Child
        Attacher.Child => Detacher.Child
        Detacher.Child => Attacher_2.Child
        ClosestObject_5.ClosestObject => Attacher_2.Parent
    - LinkTool [mechanism] at (0, 0, 0) mm, rotated rx 180 ry 0 rz 0 deg
        TCP LinkTool at (0, 0, 170) mm
        links: Tool_Link
    - ClosestObject [smart component, from Components\ClosestObject.rslib] at (-4906.26, 3034.43, -624.04) mm
        properties: ReferenceObject=Link_Tool_smart_2; ReferencePoint=[0 0 0]; RootObject=(none); ClosestObject=Wheel_tool_smart; ClosestPart=Tool_Wheel; Distance=0.444832855224609
    - Attacher [smart component, from Components\Attacher.rslib] at (-4906.26, 3034.43, -624.04) mm
        properties: Parent=Link_Tool_smart_2; Flange=0; Child=Wheel_tool_smart; Mount=false; Offset=[0 0 0]; Orientation=[0 0 0]
    - LogicGate [smart component, from Components\LogicGate.rslib] at (-4906.26, 3034.43, -624.04) mm
        properties: Operator=NOT; Delay=0
    - Detacher [smart component, from Components\Detacher.rslib] at (-4906.26, 3034.43, -624.04) mm
        properties: Child=Wheel_tool_smart; KeepPosition=true
    - Attacher_2 [smart component, from Components\Attacher.rslib] at (-4906.26, 3034.43, -624.04) mm
        properties: Parent=(none); Flange=0; Child=Wheel_tool_smart; Mount=false; Offset=[0 0 0]; Orientation=[0 0 0]
    - ClosestObject_5 [smart component, from Components\ClosestObject.rslib]
        properties: ReferenceObject=L2; ReferencePoint=[0 0 0]; RootObject=(none); ClosestObject=(none); ClosestPart=(none); Distance=0
  - toolHolder_11 [part] at (8016.5, 3102.04, 0) mm, size 200 x 350 x 600 mm
  - Pin_Tool_smart2 [smart component] at (8016.5, 3182.04, 619.8) mm
      signals: DI AttachPin, DO Pin_Attached
      connections:
        Pin_Tool_smart2.AttachPin -> ClosestObject.Execute
        ClosestObject.Executed -> Attacher.Execute
        Pin_Tool_smart2.AttachPin -> LogicGate.InputA
        LogicGate.Output -> Detacher.Execute
        Detacher.Executed -> Attacher_2.Execute
        Attacher.Executed -> Pin_Tool_smart2.Pin_Attached
        Pin_Tool_smart2.AttachPin -> ClosestObject_9.Execute
        ClosestObject.ReferenceObject => Attacher.Parent
        ClosestObject.ClosestObject => Attacher.Child
        Attacher.Child => Detacher.Child
        Detacher.Child => Attacher_2.Child
        ClosestObject_9.ClosestObject => Attacher_2.Parent
    - PinTool [mechanism] at (0, 0, 0) mm, rotated rx 180 ry 0 rz 0 deg
        TCP PinTool at (0, 0, 137.35) mm
        links: Tool_Arm_pin
    - ClosestObject [smart component, from Components\ClosestObject.rslib] at (-8688, 2695.24, -620.9) mm
        properties: ReferenceObject=Pin_Tool_smart2; ReferencePoint=[0 0 0]; RootObject=(none); ClosestObject=Axel_Tool_smart; ClosestPart=Tool_Axel_pin; Distance=0.139682907104492
    - Attacher [smart component, from Components\Attacher.rslib] at (-8688, 2695.24, -620.9) mm
        properties: Parent=Pin_Tool_smart2; Flange=0; Child=Axel_Tool_smart; Mount=false; Offset=[0 0 0]; Orientation=[0 0 0]
    - LogicGate [smart component, from Components\LogicGate.rslib] at (-8688, 2695.24, -620.9) mm
        properties: Operator=NOT; Delay=0
    - Detacher [smart component, from Components\Detacher.rslib] at (-8688, 2695.24, -620.9) mm
        properties: Child=Axel_Tool_smart; KeepPosition=true
    - Attacher_2 [smart component, from Components\Attacher.rslib] at (-8688, 2695.24, -620.9) mm
        properties: Parent=(none); Flange=0; Child=Axel_Tool_smart; Mount=false; Offset=[0 0 0]; Orientation=[0 0 0]
    - ClosestObject_9 [smart component, from Components\ClosestObject.rslib]
        properties: ReferenceObject=L2; ReferencePoint=[0 0 0]; RootObject=(none); ClosestObject=(none); ClosestPart=(none); Distance=0
  - 400_3 [part, from %ABB.RobotStudio.Models.Conveyors%\Conveyor Guide 400.rslib] at (12859.46, 3006.47, 0) mm, rotated rx 0 ry 0 rz 180 deg
  - Link_2 [part] at (13393.79, 6925.09, 489.42) mm, rotated rx 90 ry 0 rz -90 deg, size 186.8 x 62.5 x 1937.5 mm
  - Arm_pin_2 [part] at (10704.32, 2806.55, 846.28) mm, rotated rx 0 ry 0 rz 90 deg, size 126 x 162.5 x 125.8 mm
  - SpawnPin_2 [smart component] at (0, 735, 0) mm
      signals: DO volumeerkannt, DI spanw, DI diDeque
      connections:
        VolumeSensor.SensorOut -> LogicGate.InputA
        LineSensor_2.SensorOut -> LogicGate_2.InputA
        LogicGate_2.Output -> LinearMover.Execute
        Source.Executed -> Queue_2.Enqueue
        LogicGate.Output -> Source.Execute
        SpawnPin_2.diDeque -> Queue_2.Dequeue
        SpawnPin_2.spanw -> Source.Execute
        VolumeSensor.SensorOut -> SpawnPin_2.volumeerkannt
        Source.Copy => Queue_2.Back
    - Source [smart component, from Components\Source.rslib]
        properties: Source=Arm_pin_2; Copy=(none); Parent=(none); Position=[12.6 2.806547 0.846275]; Orientation=[0 0 1.5707963267949]; Transient=false; PhysicsBehavior=-1
    - Queue_2 [smart component, from Components\Queue.rslib]
        properties: Back=(none); Front=(none); Queue={1d260e56-3a9b-4089-bc8a-9b7fc13f89e8};{68ae6273-f876-46ed-a841-c22bc3c7f170}; NumberOfObjects=1
    - LinearMover [smart component, from Components\LinearMover.rslib]
        properties: Object=Queue_2; Direction=[-1 0 0]; Speed=0.5; Reference=Global; ReferenceObject=(none)
    - LineSensor_2 [smart component, from Components\LineSensor.rslib] at (6, 0, 0) mm
        properties: Start=[9.859459 1.8769 0.84]; End=[9.859459 2.2749 0.84]; Length=0.398; Radius=0.00524017467248908; Tag=(none); SensedPart=(none); SensedPoint=[0 0 0]
      - _sensorPart_ [part], size 10.5 x 398 x 10.5 mm
    - VolumeSensor [smart component, from Components\VolumeSensor.rslib]
        properties: CornerPoint=[11.617459 1.8719 0.86]; Orientation=[0 0 0]; Length=1.2; Width=0.4; Height=0.2; Tag=(none); PartialHit=true; SensedPart=(none)
      - _sensorPart_ [part], size 1200 x 400 x 200 mm
    - LogicGate [smart component, from Components\LogicGate.rslib]
        properties: Operator=NOT; Delay=0
    - LogicGate_2 [smart component, from Components\LogicGate.rslib]
        properties: Operator=NOT; Delay=0
  - SpawnLink_2 [smart component] at (10414.69, 13082, 0) mm
      signals: DO volumeerkannt, DI spanw, DI diDeque
      connections:
        VolumeSensor.SensorOut -> LogicGate.InputA
        LineSensor_2.SensorOut -> LogicGate_2.InputA
        LogicGate_2.Output -> LinearMover.Execute
        Source.Executed -> Queue_2.Enqueue
        LogicGate.Output -> Source.Execute
        SpawnLink_2.diDeque -> Queue_2.Dequeue
        SpawnLink_2.spanw -> Source.Execute
        VolumeSensor.SensorOut -> SpawnLink_2.volumeerkannt
        Source.Copy => Queue_2.Back
    - Source [smart component, from Components\Source.rslib]
        properties: Source=Link_2; Copy=(none); Parent=(none); Position=[11.5 6.925093 0.489424]; Orientation=[1.5707963267949 0 -1.5707963267949]; Transient=false; PhysicsBehavior=-1
    - Queue_2 [smart component, from Components\Queue.rslib]
        properties: Back=(none); Front=(none); Queue={1d260e56-3a9b-4089-bc8a-9b7fc13f89e8};{5a10ac6e-8e6d-4320-b1fc-87ca64eb2ab9};{339d23b8-4dd4-4c1e-9a58-b77691da5f86}; NumberOfObjects=1
    - LinearMover [smart component, from Components\LinearMover.rslib]
        properties: Object=Queue_2; Direction=[-1 0 0]; Speed=0.5; Reference=Global; ReferenceObject=(none)
    - LineSensor_2 [smart component, from Components\LineSensor.rslib] at (-7351.86, 0, -29.99) mm
        properties: Start=[5.47 -6.89178 0.5]; End=[5.47 -5.45178 0.5]; Length=1.44; Radius=0.0131004366812227; Tag=(none); SensedPart=(none); SensedPoint=[0 0 0]
      - _sensorPart_ [part], size 26.2 x 1440 x 26.2 mm
    - VolumeSensor [smart component, from Components\VolumeSensor.rslib]
        properties: CornerPoint=[0.761246486480401 -6.83178 0.45]; Orientation=[0 0 0]; Length=2; Width=1; Height=0.5; Tag=(none); PartialHit=true; SensedPart=(none)
      - _sensorPart_ [part], size 2000 x 1000 x 500 mm
    - LogicGate [smart component, from Components\LogicGate.rslib]
        properties: Operator=NOT; Delay=0
    - LogicGate_2 [smart component, from Components\LogicGate.rslib]
        properties: Operator=NOT; Delay=0
  - 1320_4800_6 [part, from %ABB.RobotStudio.Models.Conveyors%\Conveyor 1320 4800 h2.rslib] at (13264.62, 5686.22, 0) mm, rotated rx 0 ry 0 rz 180 deg
  - CowCatcher_Tool_smart [smart component]
      signals: DI Link_Attach, DO Link_is_attached
      connections:
        CowCatcher_Tool_smart.Link_Attach -> ClosestObject.Execute
        ClosestObject.Executed -> Attacher.Execute
        CowCatcher_Tool_smart.Link_Attach -> LogicGate.InputA
        LogicGate.Output -> Detacher.Execute
        Detacher.Executed -> Attacher_2.Execute
        Attacher.Executed -> CowCatcher_Tool_smart.Link_is_attached
        CowCatcher_Tool_smart.Link_Attach -> ClosestObject_6.Execute
        ClosestObject.ReferenceObject => Attacher.Parent
        ClosestObject.ClosestObject => Attacher.Child
        Attacher.Child => Detacher.Child
        Detacher.Child => Attacher_2.Child
        ClosestObject_6.ClosestObject => Attacher_2.Parent
    - ClosestObject [smart component, from Components\ClosestObject.rslib]
        properties: ReferenceObject=CowCatcher_Tool_smart; ReferencePoint=[0 0 0]; RootObject=(none); ClosestObject=Wheel_tool_smart; ClosestPart=Tool_Wheel; Distance=0.444832855224609
    - Attacher [smart component, from Components\Attacher.rslib]
        properties: Parent=CowCatcher_Tool_smart; Flange=0; Child=Wheel_tool_smart; Mount=false; Offset=[0 0 0]; Orientation=[0 0 0]
    - LogicGate [smart component, from Components\LogicGate.rslib]
        properties: Operator=NOT; Delay=0
    - Detacher [smart component, from Components\Detacher.rslib]
        properties: Child=Wheel_tool_smart; KeepPosition=true
    - Attacher_2 [smart component, from Components\Attacher.rslib]
        properties: Parent=(none); Flange=0; Child=Wheel_tool_smart; Mount=false; Offset=[0 0 0]; Orientation=[0 0 0]
    - CowCatcher_Tool [mechanism] at (4906.26, -1820.5, 629.91) mm, rotated rx 180 ry 0 rz -90 deg
        TCP CowCatcher_Tool at (0, 0, -240) mm, rotated rx 180 ry 0 rz 180 deg
        links: Tool_Cow_Catcher
    - ClosestObject_6 [smart component, from Components\ClosestObject.rslib]
        properties: ReferenceObject=L2; ReferencePoint=[0 0 0]; RootObject=(none); ClosestObject=(none); ClosestPart=(none); Distance=0
  - MoveTrain_Cow [smart component]
      signals: DI Move_to_Cow
      connections:
        MoveTrain_Cow.Move_to_Cow -> PoseMover.Execute
    - PoseMover [smart component, from Components\PoseMover.rslib]
        properties: Mechanism=ZugSchlitten; Pose=6; Duration=1
  - SpawnCow [smart component] at (10414.69, 1809, 0) mm
      signals: DO volumeerkannt, DI spanw, DI diDeque
      connections:
        VolumeSensor.SensorOut -> LogicGate.InputA
        LineSensor_2.SensorOut -> LogicGate_2.InputA
        LogicGate_2.Output -> LinearMover.Execute
        Source.Executed -> Queue_2.Enqueue
        LogicGate.Output -> Source.Execute
        SpawnCow.diDeque -> Queue_2.Dequeue
        SpawnCow.spanw -> Source.Execute
        Source.Copy => Queue_2.Back
    - Source [smart component, from Components\Source.rslib]
        properties: Source=Cow_Catcher; Copy=(none); Parent=(none); Position=[13 -3.839408 0.450441]; Orientation=[0 0 -1.5707963267949]; Transient=false; PhysicsBehavior=-1
    - Queue_2 [smart component, from Components\Queue.rslib]
        properties: Back=(none); Front=(none); Queue={1d260e56-3a9b-4089-bc8a-9b7fc13f89e8};{5a10ac6e-8e6d-4320-b1fc-87ca64eb2ab9};{339d23b8-4dd4-4c1e-9a58-b77691da5f86}; NumberOfObjects=1
    - LinearMover [smart component, from Components\LinearMover.rslib]
        properties: Object=Queue_2; Direction=[-1 0 0]; Speed=0.5; Reference=Global; ReferenceObject=(none)
    - LineSensor_2 [smart component, from Components\LineSensor.rslib] at (-7063.16, 0, 124.34) mm
        properties: Start=[5.47 -6.89178 0.5]; End=[5.47 -5.45178 0.5]; Length=1.44; Radius=0.0131004366812227; Tag=(none); SensedPart=(none); SensedPoint=[0 0 0]
      - _sensorPart_ [part], size 26.2 x 1440 x 26.2 mm
    - VolumeSensor [smart component, from Components\VolumeSensor.rslib] at (0, 200.73, 0) mm
        properties: CornerPoint=[0.761246486480401 -6.83178 0.49]; Orientation=[0 0 0]; Length=2; Width=1; Height=0.5; Tag=(none); PartialHit=true; SensedPart=(none)
      - _sensorPart_ [part], size 2000 x 1000 x 500 mm
    - LogicGate [smart component, from Components\LogicGate.rslib]
        properties: Operator=NOT; Delay=0
    - LogicGate_2 [smart component, from Components\LogicGate.rslib]
        properties: Operator=NOT; Delay=0
  - Stack_Tool_smart [smart component] at (4906.26, 3849.13, 626.19) mm
      signals: DI Link_Attach, DO Link_is_attached
      connections:
        Stack_Tool_smart.Link_Attach -> ClosestObject.Execute
        ClosestObject.Executed -> Attacher.Execute
        Stack_Tool_smart.Link_Attach -> LogicGate.InputA
        LogicGate.Output -> Detacher.Execute
        Detacher.Executed -> Attacher_2.Execute
        Attacher.Executed -> Stack_Tool_smart.Link_is_attached
        Stack_Tool_smart.Link_Attach -> ClosestObject_7.Execute
        ClosestObject.ReferenceObject => Attacher.Parent
        ClosestObject.ClosestObject => Attacher.Child
        Attacher.Child => Detacher.Child
        Detacher.Child => Attacher_2.Child
        ClosestObject_7.ClosestObject => Attacher_2.Parent
    - ClosestObject [smart component, from Components\ClosestObject.rslib] at (-4906.26, 3034.43, -624.04) mm
        properties: ReferenceObject=Stack_Tool_smart; ReferencePoint=[0 0 0]; RootObject=(none); ClosestObject=Wheel_tool_smart; ClosestPart=Tool_Wheel; Distance=0.444832855224609
    - Attacher [smart component, from Components\Attacher.rslib] at (-4906.26, 3034.43, -624.04) mm
        properties: Parent=Stack_Tool_smart; Flange=0; Child=Wheel_tool_smart; Mount=false; Offset=[0 0 0]; Orientation=[0 0 0]
    - LogicGate [smart component, from Components\LogicGate.rslib] at (-4906.26, 3034.43, -624.04) mm
        properties: Operator=NOT; Delay=0
    - Detacher [smart component, from Components\Detacher.rslib] at (-4906.26, 3034.43, -624.04) mm
        properties: Child=Wheel_tool_smart; KeepPosition=true
    - Attacher_2 [smart component, from Components\Attacher.rslib] at (-4906.26, 3034.43, -624.04) mm
        properties: Parent=(none); Flange=0; Child=Wheel_tool_smart; Mount=false; Offset=[0 0 0]; Orientation=[0 0 0]
    - Stack_Tool [mechanism] at (0, -1127.2, 9.68) mm, rotated rx 180 ry 0 rz -90 deg
        TCP Stack_Tool at (0, 875, 0) mm, rotated rx 0 ry -90 rz 90 deg
        links: Tool_Stack_tutorial
    - ClosestObject_7 [smart component, from Components\ClosestObject.rslib]
        properties: ReferenceObject=L2; ReferencePoint=[0 0 0]; RootObject=(none); ClosestObject=(none); ClosestPart=(none); Distance=0
  - SpawnStack [smart component] at (10414.69, 11182, 0) mm
      signals: DO volumeerkannt, DI spanw, DI diDeque
      connections:
        VolumeSensor.SensorOut -> LogicGate.InputA
        LineSensor_2.SensorOut -> LogicGate_2.InputA
        LogicGate_2.Output -> LinearMover.Execute
        Source.Executed -> Queue_2.Enqueue
        LogicGate.Output -> Source.Execute
        SpawnStack.diDeque -> Queue_2.Dequeue
        SpawnStack.spanw -> Source.Execute
        VolumeSensor.SensorOut -> SpawnStack.volumeerkannt
        Source.Copy => Queue_2.Back
    - Source [smart component, from Components\Source.rslib]
        properties: Source=Stack_tutorial_2; Copy=(none); Parent=(none); Position=[13 5.027585 1.315988]; Orientation=[-1.5707963267949 0 0]; Transient=false; PhysicsBehavior=-1
    - Queue_2 [smart component, from Components\Queue.rslib]
        properties: Back=(none); Front=(none); Queue={1d260e56-3a9b-4089-bc8a-9b7fc13f89e8};{5a10ac6e-8e6d-4320-b1fc-87ca64eb2ab9};{339d23b8-4dd4-4c1e-9a58-b77691da5f86}; NumberOfObjects=1
    - LinearMover [smart component, from Components\LinearMover.rslib]
        properties: Object=Queue_2; Direction=[-1 0 0]; Speed=0.5; Reference=Global; ReferenceObject=(none)
    - LineSensor_2 [smart component, from Components\LineSensor.rslib] at (-7341.86, 0, -29.99) mm
        properties: Start=[5.47 -6.89178 0.5]; End=[5.47 -5.45178 0.5]; Length=1.44; Radius=0.0131004366812227; Tag=(none); SensedPart=(none); SensedPoint=[0 0 0]
      - _sensorPart_ [part], size 26.2 x 1440 x 26.2 mm
    - VolumeSensor [smart component, from Components\VolumeSensor.rslib]
        properties: CornerPoint=[0.761246486480401 -6.83178 0.45]; Orientation=[0 0 0]; Length=2; Width=1; Height=0.5; Tag=(none); PartialHit=true; SensedPart=(none)
      - _sensorPart_ [part], size 2000 x 1000 x 500 mm
    - LogicGate [smart component, from Components\LogicGate.rslib]
        properties: Operator=NOT; Delay=0
    - LogicGate_2 [smart component, from Components\LogicGate.rslib]
        properties: Operator=NOT; Delay=0
  - MoveTrain_Home [smart component]
      signals: DI Go_to_Home, DO Home_Pos_reached, DI Reset
      connections:
        MoveTrain_Home.Go_to_Home -> PoseMover.Execute
        PoseMover.Executed -> LogicSRLatch.Set
        LogicSRLatch.Output -> MoveTrain_Home.Home_Pos_reached
        Comparer_2.Output -> MoveTrain_Home.Home_Pos_reached
        PoseMover.Executed -> Comparer_2.ValueA
        PoseMover.Executed -> LogicSRLatch.Set
        LogicSRLatch.Output -> MoveTrain_Home.Home_Pos_reached
        MoveTrain_Home.Reset -> LogicSRLatch.Reset
    - PoseMover [smart component, from Components\PoseMover.rslib]
        properties: Mechanism=ZugSchlitten; Pose=1; Duration=1
    - LogicSRLatch [smart component, from Components\LogicSRLatch.rslib]
  - MoveTrain_End [smart component]
      signals: DI Go_to_End
      connections:
        MoveTrain_End.Go_to_End -> PoseMover_2.Execute
    - PoseMover_2 [smart component, from Components\PoseMover.rslib]
        properties: Mechanism=ZugSchlitten; Pose=7; Duration=2
  - SpawnLocomotive [smart component]
      signals: DI SpawnLocomotive
      connections:
        SpawnLocomotive.SpawnLocomotive -> Source.Execute
    - Source [smart component, from Components\Source.rslib]
        properties: Source=train_body; Copy=(none); Parent=(none); Position=[-0.864085 0.35 1.462392]; Orientation=[1.5707963267949 0 1.5707963267949]; Transient=false; PhysicsBehavior=-1
  - Attach_Locomotive [smart component]
      signals: DI Attach_Locomotive
      connections:
        Attach_Locomotive.Attach_Locomotive -> ClosestObject_3.Execute
        ClosestObject_3.Executed -> Attacher.Execute
        Attach_Locomotive.Attach_Locomotive -> LogicGate.InputA
        LogicGate.Output -> Detacher.Execute
        ClosestObject_3.ClosestObject => Attacher.Child
        ClosestObject_3.ReferenceObject => Attacher.Parent
        Attacher.Child => Detacher.Child
    - Attacher [smart component, from Components\Attacher.rslib]
        properties: Parent=L2; Flange=0; Child=(none); Mount=false; Offset=[0 0 0]; Orientation=[0 0 0]
    - ClosestObject_3 [smart component, from Components\ClosestObject.rslib]
        properties: ReferenceObject=L2; ReferencePoint=[0 0 0]; RootObject=(none); ClosestObject=(none); ClosestPart=(none); Distance=0
    - Detacher [smart component, from Components\Detacher.rslib]
        properties: Child=(none); KeepPosition=true
    - LogicGate [smart component, from Components\LogicGate.rslib]
        properties: Operator=NOT; Delay=0
  - clearLocomotive [smart component]
      signals: DI clear
      connections:
        clearLocomotive.clear -> ClosestObject.Execute
        ClosestObject.Executed -> Repeater.Execute
        Repeater.Output -> ClosestObject_2.Execute
        ClosestObject_2.Executed -> Sink.Execute
        Repeater.Output -> Counter.Increase
        Comparer.Output -> Sink_2.Execute
        Sink_2.Executed -> Counter.Reset
        ClosestObject.ClosestObject => ClosestObject_2.ReferenceObject
        ClosestObject_2.ClosestObject => Sink.Object
        Counter.Count => Comparer.ValueA
        ClosestObject.ClosestObject => Sink_2.Object
    - ClosestObject [smart component, from Components\ClosestObject.rslib]
        properties: ReferenceObject=L2; ReferencePoint=[0 0 0]; RootObject=(none); ClosestObject=(none); ClosestPart=(none); Distance=0
    - Sink [smart component, from Components\Sink.rslib]
        properties: Object=(none)
    - ClosestObject_2 [smart component, from Components\ClosestObject.rslib]
        properties: ReferenceObject=(none); ReferencePoint=[0 0 0]; RootObject=(none); ClosestObject=(none); ClosestPart=(none); Distance=0
    - Repeater [smart component, from Components\Repeater.rslib]
        properties: Count=16
    - Counter [smart component, from Components\Counter.rslib]
        properties: Count=0
    - Comparer [smart component, from Components\Comparer.rslib]
        properties: ValueA=0; Operator=>=; ValueB=16
    - Sink_2 [smart component, from Components\Sink.rslib]
        properties: Object=(none)
Attachment: IRB6660_100_335__01 is attached to IRBT6004_STD_0_0_5__04 / Link1
Attachment: AttachTool_Rob1 is attached to IRB6660_100_335__01 / Link6
Attachment: AttachTool_Rob2 is attached to IRB2400_16_150__03 / Link6
Attachment: Locomotive is attached to train_body
Attachment: IRB6660_100_335__01_2 is attached to IRBT6004_STD_0_0_5__04_2 / Link1
Attachment: Link_Tool_smart_2 is attached to train_body
Collision set CollisionSet_1: Link against IRBT6004_STD_0_0_5__04, IRB2400_16_150__03, toolHolder_3, near miss 0 m
Collision set CollisionSet_2: IRB2400_16_150__03, Tool_Arm_pin, Tool_Axel_pin against 400_2, 400, Track_End, Carriage, near miss 0 m
Collision set CollisionSet_3: IRB2400_16_150__03_2, Tool_Axel_pin, Tool_Arm_pin against 400_guide, 400_3, Track_End, near miss 0 m
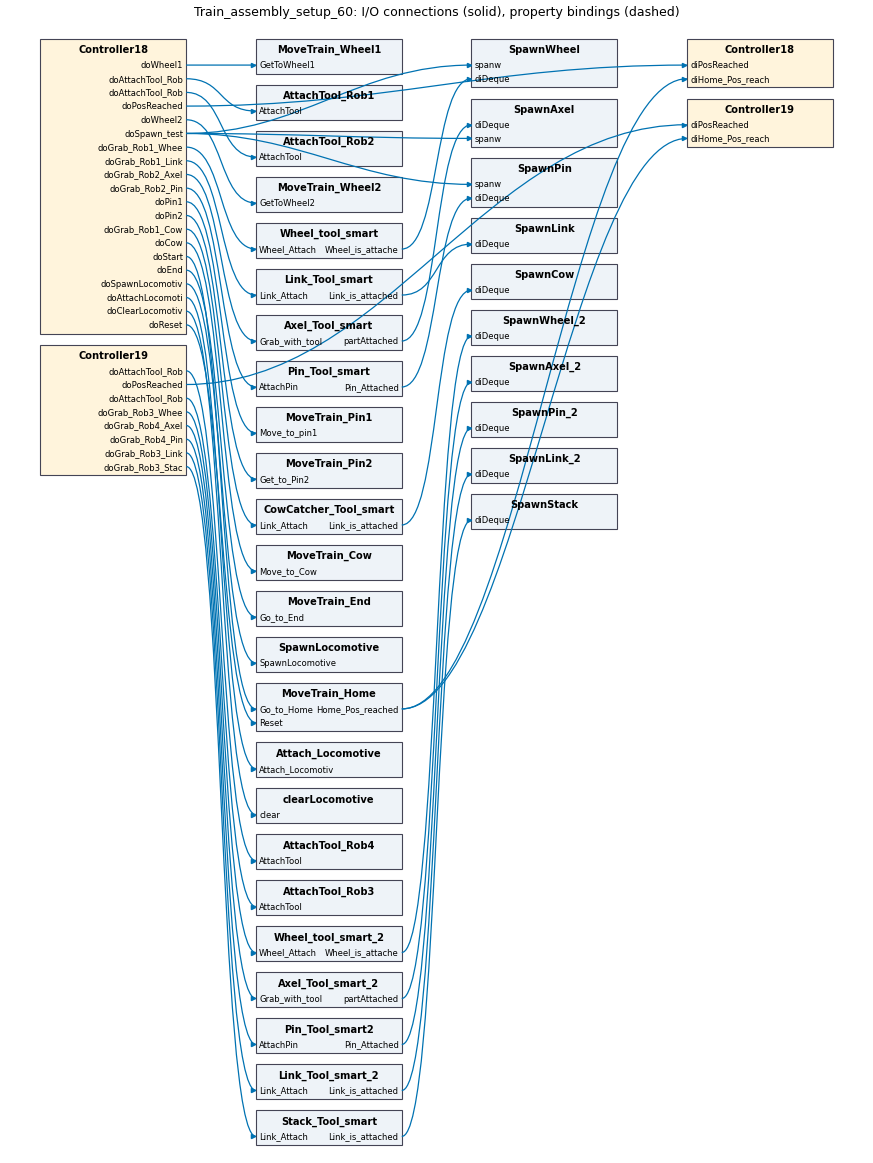
Station logic (signal -> signal, property => property):
  Controller18.doWheel1 -> MoveTrain_Wheel1.GetToWheel1
  Controller18.doAttachTool_Rob1 -> AttachTool_Rob1.AttachTool
  Controller18.doAttachTool_Rob2 -> AttachTool_Rob2.AttachTool
  Controller18.doPosReached -> Controller18.diPosReached
  Controller18.doWheel2 -> MoveTrain_Wheel2.GetToWheel2
  Controller18.doSpawn_test -> SpawnWheel.spanw
  Wheel_tool_smart.Wheel_is_attached -> SpawnWheel.diDeque
  Axel_Tool_smart.partAttached -> SpawnAxel.diDeque
  Controller18.doSpawn_test -> SpawnAxel.spanw
  Axel_Tool_smart_2.partAttached -> SpawnAxel_2.diDeque
  Controller19.doAttachTool_Rob4 -> AttachTool_Rob4.AttachTool
  Controller19.doPosReached -> Controller19.diPosReached
  Controller19.doAttachTool_Rob3 -> AttachTool_Rob3.AttachTool
  Wheel_tool_smart_2.Wheel_is_attached -> SpawnWheel_2.diDeque
  Controller18.doGrab_Rob1_Wheel -> Wheel_tool_smart.Wheel_Attach
  Controller18.doGrab_Rob1_Link -> Link_Tool_smart.Link_Attach
  Controller18.doGrab_Rob2_Axel -> Axel_Tool_smart.Grab_with_tool
  Controller18.doGrab_Rob2_Pin -> Pin_Tool_smart.AttachPin
  Controller18.doPin1 -> MoveTrain_Pin1.Move_to_pin1
  Controller18.doSpawn_test -> SpawnPin.spanw
  Pin_Tool_smart.Pin_Attached -> SpawnPin.diDeque
  Link_Tool_smart.Link_is_attached -> SpawnLink.diDeque
  Controller18.doPin2 -> MoveTrain_Pin2.Get_to_Pin2
  Controller19.doGrab_Rob3_Wheel -> Wheel_tool_smart_2.Wheel_Attach
  Controller19.doGrab_Rob4_Axel -> Axel_Tool_smart_2.Grab_with_tool
  Controller19.doGrab_Rob4_Pin -> Pin_Tool_smart2.AttachPin
  Controller19.doGrab_Rob3_Link -> Link_Tool_smart_2.Link_Attach
  Pin_Tool_smart2.Pin_Attached -> SpawnPin_2.diDeque
  Link_Tool_smart_2.Link_is_attached -> SpawnLink_2.diDeque
  Controller18.doGrab_Rob1_Cow -> CowCatcher_Tool_smart.Link_Attach
  Controller18.doCow -> MoveTrain_Cow.Move_to_Cow
  CowCatcher_Tool_smart.Link_is_attached -> SpawnCow.diDeque
  Controller19.doGrab_Rob3_Stack -> Stack_Tool_smart.Link_Attach
  Stack_Tool_smart.Link_is_attached -> SpawnStack.diDeque
  Controller18.doStart -> MoveTrain_Home.Go_to_Home
  Controller18.doEnd -> MoveTrain_End.Go_to_End
  Controller18.doSpawnLocomotive -> SpawnLocomotive.SpawnLocomotive
  Controller18.doAttachLocomotive -> Attach_Locomotive.Attach_Locomotive
  Controller18.doClearLocomotive -> clearLocomotive.clear
  MoveTrain_Home.Home_Pos_reached -> Controller18.diHome_Pos_reached
  MoveTrain_Home.Home_Pos_reached -> Controller19.diHome_Pos_reached
  Controller18.doReset -> MoveTrain_Home.Reset
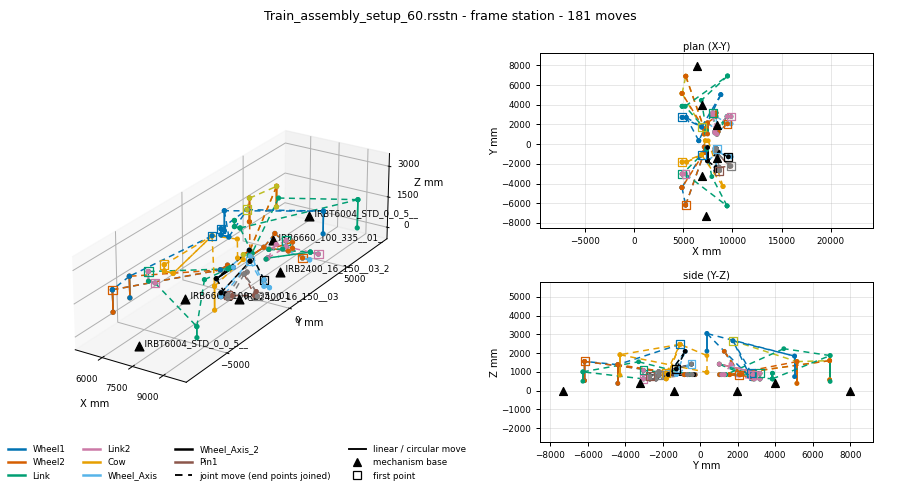
[picture p0: tool path of Train_assembly_setup_60.rsstn in frame station, 181 of 181 moves have a stored position in this frame; points joined in program order, loops and branches not executed]
Targets, tools, work objects and paths stored in the station, written as RAPID:
! task T_ROB1
MODULE Module1
  CONST robtarget Target_10:=[[5656.566354703,0,2084.5],[0.5,0,0.866025404,0],[0,0,0,0],[3495.72,9E+09,9E+09,9E+09,9E+09,9E+09]];
  CONST robtarget Target_20:=[[561.58606017,1618.325597729,146.68401849],[0,-0.707106781,0.707106781,0],[0,0,-1,0],[400,9E+09,9E+09,9E+09,9E+09,9E+09]];
  CONST robtarget Target_15:=[[562.33306017,1622.208597729,1172.76001849],[0,-0.707106781,0.707106781,0],[0,0,-1,0],[400,9E+09,9E+09,9E+09,9E+09,9E+09]];
  CONST robtarget Target_12:=[[2335.05306017,2000.172597729,-0.248],[0,-0.707106781,0.707106781,0],[1,0,0,0],[3513.18,9E+09,9E+09,9E+09,9E+09,9E+09]];
  CONST robtarget Target_11:=[[2335.05306017,2000.172597729,999.752],[0,-0.707106781,0.707106781,0],[1,0,0,0],[3513.18,9E+09,9E+09,9E+09,9E+09,9E+09]];
  CONST robtarget Target_30:=[[5889.197809027,-261.464857776,465.5],[0.5,0.5,0.5,0.5],[0,0,0,0],[3752.46,9E+09,9E+09,9E+09,9E+09,9E+09]];
  CONST robtarget Target_35:=[[6464.06006017,-261.464857776,465.5],[0.5,0.5,0.5,0.5],[0,0,0,0],[3752.46,9E+09,9E+09,9E+09,9E+09,9E+09]];
  CONST robtarget Target_45:=[[3704.62206017,1976.511597729,239.54],[0,-0.707106781,0.707106781,0],[0,0,-1,0],[3495.72,9E+09,9E+09,9E+09,9E+09,9E+09]];
  CONST robtarget Target_40:=[[3704.62206017,1976.511597729,692.082613253],[0,-0.707106781,0.707106781,0],[0,0,0,0],[3495.72,9E+09,9E+09,9E+09,9E+09,9E+09]];
  CONST robtarget Target_50:=[[3704.62206017,1640.918031273,239.54],[0,-0.707106781,0.707106781,0],[0,0,-1,0],[3495.72,9E+09,9E+09,9E+09,9E+09,9E+09]];
  CONST robtarget Target_60:=[[470.49306017,-2581.957402271,115.554],[0,0,1,0],[-2,0,-2,0],[581.02,9E+09,9E+09,9E+09,9E+09,9E+09]];
  CONST robtarget Target_55:=[[470.49306017,-2581.957402271,615.554],[0,0,1,0],[-2,0,-2,0],[581.02,9E+09,9E+09,9E+09,9E+09,9E+09]];
  CONST robtarget Target_70:=[[6153.882486876,-485.906061906,465.5],[0.707106781,0,0.707106781,0],[-1,-1,-1,0],[4071.68,9E+09,9E+09,9E+09,9E+09,9E+09]];
  CONST robtarget Target_80:=[[6330.857575887,-485.385228168,465.5],[0.707106781,0,0.707106781,0],[0,0,-1,0],[4071.68,9E+09,9E+09,9E+09,9E+09,9E+09]];
  CONST robtarget Target_56:=[[3444.659164522,-1034.307570053,1153.41849003],[0,0,1,0],[-1,-1,-1,0],[581.02,9E+09,9E+09,9E+09,9E+09,9E+09]];
  CONST robtarget Target_90:=[[4918.55506017,1976.511597729,245.412],[0,-0.707106781,0.707106781,0],[0,0,-1,0],[3495.720148087,9E+09,9E+09,9E+09,9E+09,9E+09]];
  CONST robtarget Target_85:=[[4918.55506017,1976.511597729,545.412],[0,-0.707106781,0.707106781,0],[0,0,-1,0],[3495.720148087,9E+09,9E+09,9E+09,9E+09,9E+09]];
  CONST robtarget Target_100:=[[4918.55506017,1521.254029714,245.412],[0,-0.707106781,0.707106781,0],[0,0,-1,0],[3495.720148087,9E+09,9E+09,9E+09,9E+09,9E+09]];
  CONST robtarget Target_110:=[[2449.64706017,-2170.080778234,437.993725488],[0,0.707106781,0.707106781,0],[-2,0,-1,0],[3495.720148087,9E+09,9E+09,9E+09,9E+09,9E+09]];
  CONST robtarget Target_105:=[[2449.64706017,-2170.080778234,1529.836038486],[0,0.707106781,0.707106781,0],[-2,0,-1,0],[3495.720148087,9E+09,9E+09,9E+09,9E+09,9E+09]];
  CONST robtarget Target_120:=[[7089.05506017,-380.557132001,590.500240539],[0,0.707106781,0.707106781,0],[-1,0,0,0],[4700,9E+09,9E+09,9E+09,9E+09,9E+09]];
  CONST robtarget Target_115:=[[7089.05506017,-669.254966247,590.500240539],[0,0.707106781,0.707106781,0],[-1,0,0,0],[4700,9E+09,9E+09,9E+09,9E+09,9E+09]];
  CONST robtarget Target_130:=[[7089.05506017,-369.254966247,1484.246635126],[0,0.707106781,0.707106781,0],[-1,0,0,0],[4700,9E+09,9E+09,9E+09,9E+09,9E+09]];
  PROC main()
    Reset doStart;
    Reset doClearLocomotive;
    Reset doGetLocomotive;
    Reset doAttachLocomotive;
    Reset doAttachTool_Rob1;
    Reset doPosReached;
    Reset doGrab_Rob1_Link;
    Reset doGrab_Rob1_Wheel;
    Reset doGrab_Rob1_Cow;
    Reset doSpawn_test;
    Set doSpawn_test;
    Reset doSpawn_test;
    Set doSpawnLocomotive;
    Set doAttachLocomotive;
    Reset doSpawnLocomotive;
    Set doWheel1;
    Wheel1;
    Reset doWheel1;
    Set doReset;
    Reset doReset;
    Set doWheel2;
    Wheel2;
    Reset doWheel2;
    Set doPin1;
    WaitTime 1.5;
    Reset doPin1;
    Link;
    Set doPin2;
    WaitTime 1.5;
    Reset doPin2;
    Link2;
    Cow;
    Set doEnd;
    WaitTime 2;
    Reset doEnd;
    Set doClearLocomotive;
    Reset doClearLocomotive;
    Reset doAttachLocomotive;
    Set doStart;
  ENDPROC
  PROC Wheel1()
    MoveJ Target_10,v7000,fine,tool0\WObj:=wobj0;
    MoveJ Target_11,v7000,z100,tool0\WObj:=wobj0;
    MoveL Target_12,v7000,fine,tool0\WObj:=wobj0;
    Set doAttachTool_Rob1;
    MoveL Target_11,v7000,z50,WheelTool\WObj:=wobj0;
    MoveJ Target_15,v7000,z50,WheelTool\WObj:=wobj0;
    MoveL Target_20,v7000,fine,WheelTool\WObj:=wobj0;
    SetDO doGrab_Rob1_Wheel,1;
    MoveL Target_15,v7000,z150,WheelTool\WObj:=wobj0;
    MoveJ Target_30,v7000,fine,WheelTool\WObj:=wobj0;
    Set doPosReached;
    MoveL Target_35,v7000,fine,WheelTool\WObj:=wobj0;
    WaitTime 3;
    Reset doPosReached;
    Reset doGrab_Rob1_Wheel;
    MoveL Target_30,v7000,fine,WheelTool\WObj:=wobj0;
  ENDPROC
  PROC Wheel2()
    MoveJ Target_15,v7000,z200,WheelTool\WObj:=wobj0;
    MoveL Target_20,v7000,fine,WheelTool\WObj:=wobj0;
    Set doGrab_Rob1_Wheel;
    MoveL Target_15,v7000,z200,WheelTool\WObj:=wobj0;
    MoveJ Target_30,v7000,fine,WheelTool\WObj:=wobj0;
    Set doPosReached;
    MoveL Target_35,v7000,fine,WheelTool\WObj:=wobj0;
    WaitTime 3;
    SetDO doGrab_Rob1_Wheel,0;
    Reset doPosReached;
    MoveL Target_30,v7000,z100,WheelTool\WObj:=wobj0;
    MoveJ Target_11,v7000,z100,tool0\WObj:=wobj0;
    MoveL Target_12,v7000,fine,tool0\WObj:=wobj0;
    Reset doAttachTool_Rob1;
    MoveL Target_11,v7000,fine,tool0\WObj:=wobj0;
  ENDPROC
  PROC Link()
    MoveJ Target_40,v7000,fine,tool0\WObj:=wobj0;
    MoveL Target_45,v7000,fine,tool0\WObj:=wobj0;
    Set doAttachTool_Rob1;
    MoveL Target_50,v7000,fine,tool0\WObj:=wobj0;
    MoveJ Target_55,v7000,fine,LinkTool\WObj:=wobj0;
    MoveL Target_60,v7000,fine,LinkTool\WObj:=wobj0;
    Set doGrab_Rob1_Link;
    MoveL Target_55,v7000,fine,LinkTool\WObj:=wobj0;
    MoveJ Target_56,v7000,fine,LinkTool\WObj:=wobj0;
    MoveJ Target_70,v7000,fine,LinkTool\WObj:=wobj0;
    MoveL Target_80,v7000,fine,LinkTool\WObj:=wobj0;
    Set doPosReached;
    WaitTime 4;
    Reset doGrab_Rob1_Link;
    MoveL Target_70,v7000,fine,LinkTool\WObj:=wobj0;
    MoveJ Target_40,v7000,fine,tool0\WObj:=wobj0;
  ENDPROC
  PROC Link2()
    MoveJ Target_50,v7000,fine,tool0\WObj:=wobj0;
    MoveL Target_45,v7000,fine,tool0\WObj:=wobj0;
    Reset doAttachTool_Rob1;
    MoveJ Target_40,v7000,fine,tool0\WObj:=wobj0;
  ENDPROC
  PROC Cow()
    MoveJ Target_85,v7000,fine,tool0\WObj:=wobj0;
    MoveL Target_90,v7000,fine,tool0\WObj:=wobj0;
    Set doAttachTool_Rob1;
    MoveL Target_100,v7000,fine,tool0\WObj:=wobj0;
    MoveJ Target_10,v7000,z200,CowCatcher_Tool\WObj:=wobj0;
    Set doCow;
    MoveJ Target_105,v7000,fine,CowCatcher_Tool\WObj:=wobj0;
    MoveL Target_110,v7000,fine,CowCatcher_Tool\WObj:=wobj0;
    Set doGrab_Rob1_Cow;
    Reset doCow;
    MoveL Target_105,v7000,fine,CowCatcher_Tool\WObj:=wobj0;
    MoveJ Target_115,v7000,fine,CowCatcher_Tool\WObj:=wobj0;
    MoveL Target_120,v7000,fine,CowCatcher_Tool\WObj:=wobj0;
    Reset doGrab_Rob1_Cow;
    MoveJ Target_130,v7000,fine,CowCatcher_Tool\WObj:=wobj0;
    MoveJ Target_10,v7000,z200,CowCatcher_Tool\WObj:=wobj0;
    MoveJ Target_100,v7000,fine,tool0\WObj:=wobj0;
    MoveL Target_90,v7000,fine,tool0\WObj:=wobj0;
    Reset doAttachTool_Rob1;
    MoveL Target_85,v7000,fine,tool0\WObj:=wobj0;
    MoveJ Target_10,v7000,fine,tool0\WObj:=wobj0;
  ENDPROC
ENDMODULE

! task T_ROB1
MODULE CalibData
  PERS tooldata WheelTool:=[TRUE,[[0,0,380],[1,0,0,0]],[1,[0,0,1],[1,0,0,0],0,0,0]];
  PERS tooldata LinkTool:=[TRUE,[[0,0,170],[1,0,0,0]],[1,[0,0,1],[1,0,0,0],0,0,0]];
  PERS tooldata CowCatcher_Tool:=[TRUE,[[0,0,240],[1,0,0,0]],[1,[0,0,1],[1,0,0,0],0,0,0]];
  TASK PERS wobjdata Slider:=[FALSE,TRUE,"",[[6739.06,1423.88,215.5],[0.707107,0,0,-0.707107]],[[0,0,0],[1,0,0,0]]];
ENDMODULE

! task T_ROB2
MODULE Module1
  CONST robtarget Target_10:=[[6267.490201295,-1521.467388107,1028],[0.49999984,-0.000692849,0.866025127,0.000400017],[-1,0,0,0],[9E+09,9E+09,9E+09,9E+09,9E+09,9E+09]];
  CONST robtarget Target_20:=[[4048.66106017,-1461.964402271,415.5],[0,-0.707106781,0.707106781,0],[1,0,-4,0],[9E+09,9E+09,9E+09,9E+09,9E+09,9E+09]];
  CONST robtarget Target_30:=[[4043.81506017,-1460.570402271,236.292],[0,-0.707106781,0.707106781,0],[1,0,-4,0],[9E+09,9E+09,9E+09,9E+09,9E+09,9E+09]];
  CONST robtarget Target_40:=[[4374.629364569,-1460.570402271,236.292],[0,-0.707106781,0.707106781,0],[1,0,-4,0],[9E+09,9E+09,9E+09,9E+09,9E+09,9E+09]];
  CONST robtarget Target_50:=[[5458.184389036,-2985.996683325,470.319],[0.707106781,0.707106781,0,0],[-1,-2,-2,0],[9E+09,9E+09,9E+09,9E+09,9E+09,9E+09]];
  CONST robtarget Target_45:=[[5458.184389036,-2715.030665101,470.319],[0.707106781,0.707106781,0,0],[-1,-2,-2,0],[9E+09,9E+09,9E+09,9E+09,9E+09,9E+09]];
  CONST robtarget Target_60:=[[5458.184389036,-2715.030665101,770.319],[0.707106781,0.707106781,0,0],[-1,-2,-2,0],[9E+09,9E+09,9E+09,9E+09,9E+09,9E+09]];
  CONST robtarget Target_70:=[[6401.310622675,-601.120402271,465.5],[0.5,0.5,0.5,0.5],[0,-2,-2,0],[9E+09,9E+09,9E+09,9E+09,9E+09,9E+09]];
  CONST robtarget Target_65:=[[5044.287014607,-601.120402271,465.5],[0.5,0.5,0.5,0.5],[1,-1,-2,0],[9E+09,9E+09,9E+09,9E+09,9E+09,9E+09]];
  CONST robtarget Target_80:=[[5931.283924416,-1692.54341973,1708.487037907],[0.825139706,0.151144504,-0.005175112,0.544309675],[-1,-2,-2,0],[9E+09,9E+09,9E+09,9E+09,9E+09,9E+09]];
  CONST robtarget Target_90:=[[4043.81506017,-1805.231402271,236.398],[0,-0.707106781,0.707106781,0],[-2,0,1,0],[9E+09,9E+09,9E+09,9E+09,9E+09,9E+09]];
  CONST robtarget Target_85:=[[4043.81506017,-1805.231402271,395.066903606],[0,-0.707106781,0.707106781,0],[-2,0,1,0],[9E+09,9E+09,9E+09,9E+09,9E+09,9E+09]];
  CONST robtarget Target_100:=[[4374.567164463,-1805.231402271,236.398],[0,-0.707106781,0.707106781,0],[-2,0,1,0],[9E+09,9E+09,9E+09,9E+09,9E+09,9E+09]];
  CONST robtarget Target_110:=[[4520.58906017,-2961.913402271,439.701],[0.707106781,0.707106781,0,0],[-2,1,-1,0],[9E+09,9E+09,9E+09,9E+09,9E+09,9E+09]];
  CONST robtarget Target_105:=[[4520.58906017,-2824.663402271,439.701],[0.707106781,0.707106781,0,0],[-2,1,-1,0],[9E+09,9E+09,9E+09,9E+09,9E+09,9E+09]];
  CONST robtarget Target_120:=[[4520.58906017,-2903.62720204,639.701],[0.707106781,0.707106781,0,0],[-2,1,-1,0],[9E+09,9E+09,9E+09,9E+09,9E+09,9E+09]];
  CONST robtarget Target_130:=[[6299.812010333,-1352.722903469,465.5],[0.5,0.5,0.5,0.5],[0,-2,-2,0],[9E+09,9E+09,9E+09,9E+09,9E+09,9E+09]];
  CONST robtarget Target_125:=[[6062.74483872,-1352.722903469,465.5],[0.5,0.5,0.5,0.5],[0,-2,-2,0],[9E+09,9E+09,9E+09,9E+09,9E+09,9E+09]];
  PROC main()
    Reset doGrab_Rob2_Axel;
    Reset doGrab_Rob2_Pin;
    Reset doAttachTool_Rob2;
    Wheel_Axis;
    Wheel_Axis_2;
    WaitTime 1.5;
    Pin1;
    Pin2;
  ENDPROC
  PROC Wheel_Axis()
    MoveJ Target_10,v7000,fine,tool0\WObj:=wobj0;
    MoveJ Target_20,v7000,fine,tool0\WObj:=wobj0;
    MoveL Target_30,v7000,fine,tool0\WObj:=wobj0;
    SetDO doAttachTool_Rob2,1;
    MoveL Target_40,v7000,fine,tool0\WObj:=wobj0;
    MoveJ Target_10,v7000,z40,AxelTool\WObj:=wobj0;
    MoveJ Target_45,v7000,fine,AxelTool\WObj:=wobj0;
    MoveL Target_50,v7000,fine,AxelTool\WObj:=wobj0;
    Set doGrab_Rob2_Axel;
    MoveL Target_60,v7000,z100,AxelTool\WObj:=wobj0;
    MoveJ Target_80,v7000,z200,AxelTool\WObj:=wobj0;
    MoveJ Target_65,v7000,z100,AxelTool\WObj:=wobj0;
    MoveL Target_70,v7000,fine,AxelTool\WObj:=wobj0;
    Reset doGrab_Rob2_Axel;
    MoveL Target_65,v7000,z150,AxelTool\WObj:=wobj0;
    MoveJ Target_80,v7000,z150,AxelTool\WObj:=wobj0;
    MoveJ Target_45,v7000,fine,AxelTool\WObj:=wobj0;
    MoveL Target_50,v7000,fine,AxelTool\WObj:=wobj0;
  ENDPROC
  PROC Wheel_Axis_2()
    Set doGrab_Rob2_Axel;
    MoveL Target_60,v7000,z100,AxelTool\WObj:=wobj0;
    MoveJ Target_80,v7000,z50,AxelTool\WObj:=wobj0;
    MoveJ Target_65,v7000,z80,AxelTool\WObj:=wobj0;
    MoveL Target_70,v7000,fine,AxelTool\WObj:=wobj0;
    Reset doGrab_Rob2_Axel;
    MoveL Target_65,v7000,z200,AxelTool\WObj:=wobj0;
    MoveJ Target_40,v7000,fine,tool0\WObj:=wobj0;
    MoveL Target_30,v7000,fine,tool0\WObj:=wobj0;
    Reset doAttachTool_Rob2;
    MoveL Target_20,v7000,z50,tool0\WObj:=wobj0;
    MoveJ Target_10,v7000,fine,tool0\WObj:=wobj0;
  ENDPROC
  PROC Pin1()
    MoveJ Target_85,v7000,fine,tool0\WObj:=wobj0;
    MoveL Target_90,v7000,fine,tool0\WObj:=wobj0;
    Set doAttachTool_Rob2;
    MoveL Target_100,v7000,fine,tool0\WObj:=wobj0;
    MoveJ Target_105,v7000,fine,PinTool\WObj:=wobj0;
    MoveL Target_110,v7000,fine,PinTool\WObj:=wobj0;
    Set doGrab_Rob2_Pin;
    MoveL Target_120,v7000,fine,PinTool\WObj:=wobj0;
    MoveJ Target_125,v7000,fine,PinTool\WObj:=wobj0;
    MoveL Target_130,v7000,fine,PinTool\WObj:=wobj0;
    Reset doGrab_Rob2_Pin;
    MoveL Target_125,v7000,fine,PinTool\WObj:=wobj0;
    MoveJ Target_105,v7000,fine,PinTool\WObj:=wobj0;
    WaitTime 2;
  ENDPROC
  PROC Pin2()
    MoveL Target_110,v7000,fine,PinTool\WObj:=wobj0;
    Set doGrab_Rob2_Pin;
    MoveL Target_120,v7000,fine,PinTool\WObj:=wobj0;
    MoveJ Target_125,v7000,fine,PinTool\WObj:=wobj0;
    MoveL Target_130,v7000,fine,PinTool\WObj:=wobj0;
    Reset doGrab_Rob2_Pin;
    MoveL Target_125,v7000,fine,PinTool\WObj:=wobj0;
    MoveJ Target_100,v7000,fine,tool0\WObj:=wobj0;
    MoveL Target_90,v7000,fine,tool0\WObj:=wobj0;
    Reset doAttachTool_Rob2;
    MoveL Target_85,v7000,fine,tool0\WObj:=wobj0;
    MoveJ Target_10,v7000,fine,tool0\WObj:=wobj0;
  ENDPROC
ENDMODULE

! task T_ROB2
MODULE CalibData
  PERS tooldata AxelTool:=[TRUE,[[0,0,262.487],[1,0,0,0]],[1,[0,0,1],[1,0,0,0],0,0,0]];
  PERS tooldata PinTool:=[TRUE,[[0,0,137.349],[1,0,0,0]],[1,[0,0,1],[1,0,0,0],0,0,0]];
  TASK PERS wobjdata Slider:=[FALSE,TRUE,"",[[6739.06,1423.88,215.5],[0.707107,0,0,-0.707107]],[[0,0,0],[1,0,0,0]]];
ENDMODULE

! task T_ROB1
MODULE Module1
  CONST robtarget Target_10:=[[5656.215997788,0,2274.5],[0.5,0,0.866025404,0],[0,0,0,0],[3427.51,9E+09,9E+09,9E+09,9E+09,9E+09]];
  CONST robtarget Target_20:=[[2244.163836229,-1985.634674649,-0.248],[0,0.707106781,0.707106781,0],[-2,0,-1,0],[3427.51,9E+09,9E+09,9E+09,9E+09,9E+09]];
  CONST robtarget Target_15:=[[2244.163836229,-1985.634674649,1162.636316554],[0,0.707106781,0.707106781,0],[-2,0,-1,0],[3427.51,9E+09,9E+09,9E+09,9E+09,9E+09]];
  CONST robtarget Target_30:=[[496.303836229,-1607.890573206,190.951082311],[0,0.707106781,0.707106781,0],[-2,0,-1,0],[216.1,9E+09,9E+09,9E+09,9E+09,9E+09]];
  CONST robtarget Target_25:=[[496.303836229,-1607.890573206,1213.950662918],[0,0.707106781,0.707106781,0],[-2,0,-1,0],[216.1,9E+09,9E+09,9E+09,9E+09,9E+09]];
  CONST robtarget Target_40:=[[5838.630384805,261.678430529,465.5],[0.5,-0.5,0.5,-0.5],[0,-2,0,0],[3427.51,9E+09,9E+09,9E+09,9E+09,9E+09]];
  CONST robtarget Target_45:=[[6375.465364122,261.678430529,465.5],[0.5,-0.5,0.5,-0.5],[0,-2,0,0],[3427.51,9E+09,9E+09,9E+09,9E+09,9E+09]];
  CONST robtarget Target_55:=[[3547.028836229,-1973.768674649,241.691],[0,0.707106781,0.707106781,0],[-1,0,0,0],[3427.510261536,9E+09,9E+09,9E+09,9E+09,9E+09]];
  CONST robtarget Target_50:=[[3547.028836229,-1973.768674649,541.691],[0,0.707106781,0.707106781,0],[-1,0,0,0],[3427.510261536,9E+09,9E+09,9E+09,9E+09,9E+09]];
  CONST robtarget Target_60:=[[3547.028836229,-1673.768674649,241.691],[0,0.707106781,0.707106781,0],[-1,0,0,0],[3427.510261536,9E+09,9E+09,9E+09,9E+09,9E+09]];
  CONST robtarget Target_65:=[[471.065836229,2633.953325351,104.924],[0,0,1,0],[1,0,1,0],[896.78,9E+09,9E+09,9E+09,9E+09,9E+09]];
  CONST robtarget Target_61:=[[471.065836229,2633.953325351,1485.237358833],[0,0,1,0],[1,0,1,0],[896.78,9E+09,9E+09,9E+09,9E+09,9E+09]];
  CONST robtarget Target_70:=[[6295.319802939,495.47938561,465.5],[0.707106781,0,0.707106781,0],[0,2,-3,0],[3165.71,9E+09,9E+09,9E+09,9E+09,9E+09]];
  CONST robtarget Target_67:=[[6040.233294854,495.47938561,465.5],[0.707106781,0,0.707106781,0],[-1,1,-2,0],[3165.71,9E+09,9E+09,9E+09,9E+09,9E+09]];
  CONST robtarget Target_66:=[[2944.094746015,-32.124461483,1851.04872557],[0.707106781,0,0.707106781,0],[-1,1,-2,0],[896.78,9E+09,9E+09,9E+09,9E+09,9E+09]];
  CONST robtarget Target_80:=[[4674.232836229,-1973.768674649,251.367],[0,0,1,0],[-1,2,-3,0],[3427.509307861,9E+09,9E+09,9E+09,9E+09,9E+09]];
  CONST robtarget Target_75:=[[4674.232836229,-1973.768674649,551.367],[0,0,1,0],[-1,2,-2,0],[3427.509307861,9E+09,9E+09,9E+09,9E+09,9E+09]];
  CONST robtarget Target_90:=[[4674.232836229,-1559.241103171,251.367],[0,0,1,0],[-1,2,-3,0],[3427.509307861,9E+09,9E+09,9E+09,9E+09,9E+09]];
  CONST robtarget Target_100:=[[2368.573836229,1948.831325351,1456.748561707],[0,0,1,0],[1,-2,-2,0],[3427.509307861,9E+09,9E+09,9E+09,9E+09,9E+09]];
  CONST robtarget Target_110:=[[2368.573836229,1948.831325351,362.359823755],[0,0,1,0],[1,-2,-2,0],[3427.509307861,9E+09,9E+09,9E+09,9E+09,9E+09]];
  CONST robtarget Target_120:=[[7046.158836229,-285.548674649,1722.512176943],[0.707106781,0,0,-0.707106781],[-1,-1,-1,0],[4684.15,9E+09,9E+09,9E+09,9E+09,9E+09]];
  CONST robtarget Target_115:=[[7046.158836229,-285.548674649,2659.970810566],[0.707106781,0,0,-0.707106781],[-1,-1,-1,0],[4684.15,9E+09,9E+09,9E+09,9E+09,9E+09]];
  PROC main()
    Reset doAttachTool_Rob3;
    Reset doAttachTool_Rob4;
    Reset doGrab_Rob3_Link;
    Reset doGrab_Rob3_Wheel;
    Reset doGrab_Rob3_Stack;
    Reset doGrab_Rob4_Axel;
    Reset doGrab_Rob4_Pin;
    Reset doPosReached;
    Wheel2;
    WaitTime 1.5;
    Link;
    Stack;
    Wheel;
  ENDPROC
  PROC Wheel()
    MoveJ Target_10,v7000,fine,tool0\WObj:=wobj0;
    MoveJ Target_15,v7000,z100,tool0\WObj:=wobj0;
    MoveL Target_20,v7000,fine,tool0\WObj:=wobj0;
    Set doAttachTool_Rob3;
    MoveJ Target_15,v7000,z80,WheelTool\WObj:=wobj0;
    MoveJ Target_25,v7000,z50,WheelTool\WObj:=wobj0;
    MoveL Target_30,v7000,fine,WheelTool\WObj:=wobj0;
    Set doGrab_Rob3_Wheel;
    MoveL Target_25,v7000,z150,WheelTool\WObj:=wobj0;
    MoveJ Target_40,v7000,fine,WheelTool\WObj:=wobj0;
    Set doPosReached;
    MoveL Target_45,v7000,fine,WheelTool\WObj:=wobj0;
    WaitTime 3;
    Reset doPosReached;
    Reset doGrab_Rob3_Wheel;
    MoveL Target_40,v7000,fine,WheelTool\WObj:=wobj0;
  ENDPROC
  PROC Wheel2()
    MoveJ Target_25,v7000,z100,WheelTool\WObj:=wobj0;
    MoveL Target_30,v7000,fine,WheelTool\WObj:=wobj0;
    Set doGrab_Rob3_Wheel;
    MoveL Target_25,v7000,z200,WheelTool\WObj:=wobj0;
    MoveJ Target_40,v7000,fine,WheelTool\WObj:=wobj0;
    Set doPosReached;
    MoveL Target_45,v7000,fine,WheelTool\WObj:=wobj0;
    WaitTime 3;
    Reset doPosReached;
    Reset doGrab_Rob3_Wheel;
    MoveJ Target_40,v7000,z200,WheelTool\WObj:=wobj0;
    MoveJ Target_15,v7000,z100,WheelTool\WObj:=wobj0;
    MoveL Target_20,v7000,fine,tool0\WObj:=wobj0;
    Reset doAttachTool_Rob3;
    MoveL Target_15,v7000,fine,WheelTool\WObj:=wobj0;
  ENDPROC
  PROC Link()
    MoveJ Target_50,v7000,fine,tool0\WObj:=wobj0;
    MoveJ Target_55,v7000,fine,tool0\WObj:=wobj0;
    Set doAttachTool_Rob3;
    MoveJ Target_60,v7000,fine,tool0\WObj:=wobj0;
    MoveJ Target_61,v7000,fine,LinkTool\WObj:=wobj0;
    MoveL Target_65,v7000,fine,LinkTool\WObj:=wobj0;
    Set doGrab_Rob3_Link;
    MoveL Target_61,v7000,fine,LinkTool\WObj:=wobj0;
    MoveJ Target_66,v7000,fine,tool0\WObj:=wobj0;
    MoveJ Target_67,v7000,fine,LinkTool\WObj:=wobj0;
    MoveJ Target_70,v7000,fine,LinkTool\WObj:=wobj0;
    Set doPosReached;
    WaitTime 4;
    Reset doPosReached;
    Reset doGrab_Rob3_Link;
    MoveL Target_67,v7000,fine,LinkTool\WObj:=wobj0;
    MoveJ Target_60,v7000,fine,tool0\WObj:=wobj0;
    MoveL Target_55,v7000,fine,tool0\WObj:=wobj0;
    Reset doAttachTool_Rob3;
    MoveL Target_50,v7000,fine,tool0\WObj:=wobj0;
  ENDPROC
  PROC Stack()
    MoveJ Target_75,v7000,fine,tool0\WObj:=wobj0;
    MoveL Target_80,v7000,fine,tool0\WObj:=wobj0;
    Set doAttachTool_Rob3;
    MoveL Target_90,v7000,fine,tool0\WObj:=wobj0;
    MoveJ Target_10,v7000,z200,Stack_Tool\WObj:=wobj0;
    MoveJ Target_100,v7000,fine,Stack_Tool\WObj:=wobj0;
    MoveL Target_110,v7000,fine,Stack_Tool\WObj:=wobj0;
    Set doGrab_Rob3_Stack;
    MoveL Target_100,v7000,fine,Stack_Tool\WObj:=wobj0;
    MoveJ Target_115,v7000,fine,Stack_Tool\WObj:=wobj0;
    MoveL Target_120,v7000,fine,Stack_Tool\WObj:=wobj0;
    Reset doGrab_Rob3_Stack;
    MoveL Target_115,v7000,fine,Stack_Tool\WObj:=wobj0;
    MoveJ Target_90,v7000,fine,tool0\WObj:=wobj0;
    MoveL Target_80,v7000,fine,tool0\WObj:=wobj0;
    Reset doAttachTool_Rob3;
    MoveJ Target_75,v7000,fine,tool0\WObj:=wobj0;
    MoveJ Target_10,v7000,fine,tool0\WObj:=wobj0;
  ENDPROC
ENDMODULE

! task T_ROB1
MODULE CalibData
  PERS tooldata WheelTool:=[TRUE,[[0,0,0],[1,0,0,0]],[1,[0,0,0.001],[1,0,0,0],0,0,0]];
  PERS tooldata LinkTool:=[TRUE,[[0,0,170],[1,0,0,0]],[1,[0,0,1],[1,0,0,0],0,0,0]];
  PERS tooldata Stack_Tool:=[TRUE,[[0,-50,519.006],[0.707107,0.707107,0,0]],[1,[0,0,1],[1,0,0,0],0,0,0]];
ENDMODULE

! task T_ROB2
MODULE Module1
  CONST robtarget Target_10:=[[6386.058671067,1558.823208427,1028],[0.499999547,0.001166321,0.866024618,-0.000673375],[-1,0,-1,0],[9E+09,9E+09,9E+09,9E+09,9E+09,9E+09]];
  CONST robtarget Target_20:=[[4216.565836229,1463.313325351,236.292],[0,0.707106781,0.707106781,0],[-2,0,-1,0],[9E+09,9E+09,9E+09,9E+09,9E+09,9E+09]];
  CONST robtarget Target_15:=[[4216.565836229,1463.313325351,536.292],[0,0.707106781,0.707106781,0],[-2,0,-1,0],[9E+09,9E+09,9E+09,9E+09,9E+09,9E+09]];
  CONST robtarget Target_30:=[[4571.129291705,1463.313325351,236.292],[0,0.707106781,0.707106781,0],[-2,0,-1,0],[9E+09,9E+09,9E+09,9E+09,9E+09,9E+09]];
  CONST robtarget Target_40:=[[5325.007836229,2983.750325351,470.319],[0.707106781,-0.707106781,0,0],[1,-2,0,0],[9E+09,9E+09,9E+09,9E+09,9E+09,9E+09]];
  CONST robtarget Target_50:=[[6118.131689086,1695.286342351,1708.487038],[0.845915077,-0.098816365,0.114484799,-0.511425694],[0,-2,1,0],[9E+09,9E+09,9E+09,9E+09,9E+09,9E+09]];
  CONST robtarget Target_60:=[[5230.253444265,603.868325351,465.5],[0.5,-0.5,0.5,-0.5],[-2,0,1,0],[9E+09,9E+09,9E+09,9E+09,9E+09,9E+09]];
  CONST robtarget Target_70:=[[6357.650127052,603.868325351,465.5],[0.5,-0.5,0.5,-0.5],[-1,1,1,0],[9E+09,9E+09,9E+09,9E+09,9E+09,9E+09]];
  CONST robtarget Target_35:=[[5325.007836229,2626.885237246,470.319],[0.707106781,-0.707106781,0,0],[1,-2,0,0],[9E+09,9E+09,9E+09,9E+09,9E+09,9E+09]];
  CONST robtarget Target_80:=[[4214.117836229,1136.471325351,235.299],[0,0.707106781,0.707106781,0],[-2,0,-1,0],[9E+09,9E+09,9E+09,9E+09,9E+09,9E+09]];
  CONST robtarget Target_75:=[[4214.117836229,1136.471325351,535.299],[0,0.707106781,0.707106781,0],[-2,0,-1,0],[9E+09,9E+09,9E+09,9E+09,9E+09,9E+09]];
  CONST robtarget Target_90:=[[4514.117836229,1136.471325351,235.299],[0,0.707106781,0.707106781,0],[-2,0,-1,0],[9E+09,9E+09,9E+09,9E+09,9E+09,9E+09]];
  CONST robtarget Target_100:=[[4589.611836229,2989.400325351,461.775],[0.707106781,-0.707106781,0,0],[1,-2,0,0],[9E+09,9E+09,9E+09,9E+09,9E+09,9E+09]];
  CONST robtarget Target_95:=[[4589.611836229,2589.400325351,461.775],[0.707106781,-0.707106781,0,0],[1,-2,0,0],[9E+09,9E+09,9E+09,9E+09,9E+09,9E+09]];
  CONST robtarget Target_110:=[[6253.25460644,1342.791769351,465.5],[0.5,0.5,0.5,0.5],[-1,1,-1,0],[9E+09,9E+09,9E+09,9E+09,9E+09,9E+09]];
  CONST robtarget Target_105:=[[6122.723568182,1342.791769351,465.5],[0.5,0.5,0.5,0.5],[-1,1,-1,0],[9E+09,9E+09,9E+09,9E+09,9E+09,9E+09]];
  CONST robtarget Target_120:=[[5765.937154312,1558.823208427,1028],[0.499999547,0.001166321,0.866024618,-0.000673375],[-1,0,-1,0],[9E+09,9E+09,9E+09,9E+09,9E+09,9E+09]];
  PROC main()
    Reset doAttachTool_Rob4;
    Wheel_Axis;
    Wheel_Axis2;
    WaitTime 1.5;
    Pin;
    PIn2;
  ENDPROC
  PROC Wheel_Axis()
    MoveJ Target_10,v7000,fine,tool0\WObj:=wobj0;
    MoveJ Target_15,v7000,fine,tool0\WObj:=wobj0;
    MoveL Target_20,v7000,fine,tool0\WObj:=wobj0;
    Set doAttachTool_Rob4;
    MoveL Target_30,v7000,fine,AxelTool\WObj:=wobj0;
    MoveJ Target_35,v7000,fine,AxelTool\WObj:=wobj0;
    MoveL Target_40,v7000,fine,AxelTool\WObj:=wobj0;
    Set doGrab_Rob4_Axel;
    MoveL Target_35,v7000,z100,AxelTool\WObj:=wobj0;
    MoveJ Target_50,v7000,z200,AxelTool\WObj:=wobj0;
    MoveJ Target_60,v7000,z200,AxelTool\WObj:=wobj0;
    MoveL Target_70,v7000,fine,AxelTool\WObj:=wobj0;
    Reset doGrab_Rob4_Axel;
    MoveL Target_60,v7000,z200,AxelTool\WObj:=wobj0;
    MoveJ Target_50,v7000,z200,AxelTool\WObj:=wobj0;
    MoveJ Target_35,v7000,z100,AxelTool\WObj:=wobj0;
    MoveL Target_40,v7000,fine,AxelTool\WObj:=wobj0;
  ENDPROC
  PROC Wheel_Axis2()
    Set doGrab_Rob4_Axel;
    MoveL Target_35,v7000,z100,AxelTool\WObj:=wobj0;
    MoveJ Target_50,v7000,z200,AxelTool\WObj:=wobj0;
    MoveJ Target_60,v7000,z200,AxelTool\WObj:=wobj0;
    MoveL Target_70,v7000,fine,AxelTool\WObj:=wobj0;
    Reset doGrab_Rob4_Axel;
    MoveL Target_60,v7000,z200,AxelTool\WObj:=wobj0;
    MoveJ Target_30,v7000,z100,AxelTool\WObj:=wobj0;
    MoveL Target_20,v7000,fine,tool0\WObj:=wobj0;
    Reset doAttachTool_Rob4;
    MoveL Target_15,v7000,fine,tool0\WObj:=wobj0;
    MoveJ Target_10,v7000,fine,tool0\WObj:=wobj0;
  ENDPROC
  PROC Pin()
    MoveJ Target_75,v7000,fine,tool0\WObj:=wobj0;
    MoveL Target_80,v7000,fine,tool0\WObj:=wobj0;
    Set doAttachTool_Rob4;
    MoveL Target_90,v7000,fine,tool0\WObj:=wobj0;
    MoveJ Target_10,v7000,fine,PinTool\WObj:=wobj0;
    MoveJ Target_95,v7000,z100,PinTool\WObj:=wobj0;
    MoveL Target_100,v7000,fine,PinTool\WObj:=wobj0;
    Set doGrab_Rob4_Pin;
    MoveL Target_95,v7000,z50,PinTool\WObj:=wobj0;
    MoveJ Target_105,v7000,fine,PinTool\WObj:=wobj0;
    MoveL Target_110,v7000,fine,PinTool\WObj:=wobj0;
    Reset doGrab_Rob4_Pin;
    MoveL Target_105,v7000,fine,PinTool\WObj:=wobj0;
    MoveJ Target_95,v7000,fine,PinTool\WObj:=wobj0;
    WaitTime 2;
  ENDPROC
  PROC PIn2()
    MoveL Target_100,v7000,fine,PinTool\WObj:=wobj0;
    Set doGrab_Rob4_Pin;
    MoveL Target_95,v7000,fine,PinTool\WObj:=wobj0;
    MoveJ Target_120,v7000,z100,PinTool\WObj:=wobj0;
    MoveJ Target_105,v7000,fine,PinTool\WObj:=wobj0;
    MoveL Target_110,v7000,fine,PinTool\WObj:=wobj0;
    Reset doGrab_Rob4_Pin;
    MoveL Target_105,v7000,fine,PinTool\WObj:=wobj0;
    MoveJ Target_90,v7000,fine,tool0\WObj:=wobj0;
    MoveL Target_80,v7000,fine,tool0\WObj:=wobj0;
    Reset doAttachTool_Rob4;
    MoveL Target_75,v7000,fine,tool0\WObj:=wobj0;
    MoveJ Target_10,v7000,fine,tool0\WObj:=wobj0;
  ENDPROC
ENDMODULE

! task T_ROB2
MODULE CalibData
  PERS tooldata AxelTool:=[TRUE,[[0,0,0],[1,0,0,0]],[1,[0,0,0.001],[1,0,0,0],0,0,0]];
  PERS tooldata PinTool:=[TRUE,[[0,0,137.349],[1,0,0,0]],[1,[0,0,1],[1,0,0,0],0,0,0]];
ENDMODULE

